LIN {X 0,Y 185.932,Z 327.325,A -85,B 0,C 180,E1 -22223.49,E2 -22223.49} C_VEL
LIN {X 0,Y 186.378,Z 327.271,A -85,B 0,C 180,E1 -22230.001,E2 -22230.001} C_VEL
LIN {X 0,Y 185.926,Z 327.327,A -85,B 0,C 180,E1 -22236.513,E2 -22236.513} C_VEL
LIN {X 0,Y 185.869,Z 327.333,A -85,B 0,C 180,E1 -22239.922,E2 -22239.922} C_VEL
LIN {X 0,Y 186.977,Z 330.337,A -85,B 0,C 180,E1 -22240.252,E2 -22240.252} C_VEL
LIN {X 0,Y 196.762,Z 352.168,A -85,B 0,C 180,E1 -22242.755,E2 -22242.755} C_VEL
LIN {X 0,Y 202.27,Z 367.616,A -85,B 0,C 180,E1 -22244.204,E2 -22244.204} C_VEL
LIN {X 0,Y 202.12,Z 374.541,A -85,B 0,C 180,E1 -22244.511,E2 -22244.511} C_VEL
LIN {X 0,Y 199.034,Z 429.376,A -85,B 0,C 180,E1 -22246.777,E2 -22246.777} C_VEL
LIN {X 0,Y 197.747,Z 443.213,A -85,B 0,C 180,E1 -22247.759,E2 -22247.759} C_VEL
LIN {X 0,Y 196.286,Z 455.635,A -85,B 0,C 180,E1 -22249.053,E2 -22249.053} C_VEL
LIN {X 0,Y 194.468,Z 467.347,A -85,B 0,C 180,E1 -22250.675,E2 -22250.675} C_VEL
LIN {X 0,Y 192.408,Z 479.143,A -85,B 0,C 180,E1 -22252.786,E2 -22252.786} C_VEL
LIN {X 0,Y 190.451,Z 489.318,A -85,B 0,C 180,E1 -22255.112,E2 -22255.112} C_VEL
LIN {X 0,Y 188.356,Z 499.162,A -85,B 0,C 180,E1 -22257.925,E2 -22257.925} C_VEL
LIN {X 0,Y 186.543,Z 507.642,A -85,B 0,C 180,E1 -22260.964,E2 -22260.964} C_VEL
LIN {X 0,Y 185.14,Z 514.465,A -85,B 0,C 180,E1 -22264.04,E2 -22264.04} C_VEL
LIN {X 0,Y 184.09,Z 520.754,A -85,B 0,C 180,E1 -22267.651,E2 -22267.651} C_VEL
LIN {X 0,Y 183.278,Z 524.854,A -85,B 0,C 180,E1 -22270.685,E2 -22270.685} C_VEL
LIN {X 0,Y 182.827,Z 528.069,A -85,B 0,C 180,E1 -22273.785,E2 -22273.785} C_VEL
LIN {X 0,Y 182.741,Z 530.438,A -85,B 0,C 180,E1 -22276.948,E2 -22276.948} C_VEL
LIN {X 0,Y 182.953,Z 531.969,A -85,B 0,C 180,E1 -22280.202,E2 -22280.202} C_VEL
LIN {X 0,Y 183.589,Z 532.61,A -85,B 0,C 180,E1 -22283.506,E2 -22283.506} C_VEL
LIN {X 0,Y 185.064,Z 532.068,A -85,B 0,C 180,E1 -22287.881,E2 -22287.881} C_VEL
LIN {X 0,Y 186.497,Z 530.891,A -85,B 0,C 180,E1 -22290.665,E2 -22290.665} C_VEL
LIN {X 0,Y 189.251,Z 527.772,A -85,B 0,C 180,E1 -22294.811,E2 -22294.811} C_VEL
LIN {X 0,Y 192.716,Z 523.296,A -85,B 0,C 180,E1 -22298.611,E2 -22298.611} C_VEL
LIN {X 0,Y 196.243,Z 518.203,A -85,B 0,C 180,E1 -22301.709,E2 -22301.709} C_VEL
LIN {X 0,Y 200.327,Z 511.596,A -85,B 0,C 180,E1 -22304.744,E2 -22304.744} C_VEL
LIN {X 0,Y 205.082,Z 503.165,A -85,B 0,C 180,E1 -22307.699,E2 -22307.699} C_VEL
LIN {X 0,Y 209.405,Z 494.509,A -85,B 0,C 180,E1 -22310.053,E2 -22310.053} C_VEL
LIN {X 0,Y 213.974,Z 483.997,A -85,B 0,C 180,E1 -22312.253,E2 -22312.253} C_VEL
LIN {X 0,Y 217.979,Z 473.293,A -85,B 0,C 180,E1 -22313.986,E2 -22313.986} C_VEL
LIN {X 0,Y 221.603,Z 461.549,A -85,B 0,C 180,E1 -22315.452,E2 -22315.452} C_VEL
LIN {X 0,Y 224.7,Z 448.564,A -85,B 0,C 180,E1 -22316.683,E2 -22316.683} C_VEL
LIN {X 0,Y 226.822,Z 436.927,A -85,B 0,C 180,E1 -22317.465,E2 -22317.465} C_VEL
LIN {X 0,Y 228.488,Z 423.317,A -85,B 0,C 180,E1 -22318.057,E2 -22318.057} C_VEL
LIN {X 0,Y 231.675,Z 389.447,A -85,B 0,C 180,E1 -22319.266,E2 -22319.266} C_VEL
LIN {X 0,Y 228.046,Z 381.272,A -85,B 0,C 180,E1 -22321.321,E2 -22321.321} C_VEL
LIN {X 0,Y 223.31,Z 372.435,A -85,B 0,C 180,E1 -22324.297,E2 -22324.297} C_VEL
LIN {X 0,Y 221.558,Z 369.535,A -85,B 0,C 180,E1 -22325.549,E2 -22325.549} C_VEL
LIN {X 0,Y 219.232,Z 366.365,A -85,B 0,C 180,E1 -22327.272,E2 -22327.272} C_VEL
LIN {X 0,Y 216.775,Z 362.911,A -85,B 0,C 180,E1 -22329.412,E2 -22329.412} C_VEL
LIN {X 0,Y 215.973,Z 361.635,A -85,B 0,C 180,E1 -22330.212,E2 -22330.212} C_VEL
LIN {X 0,Y 213.658,Z 358.637,A -85,B 0,C 180,E1 -22332.793,E2 -22332.793} C_VEL
LIN {X 0,Y 212.698,Z 357.131,A -85,B 0,C 180,E1 -22334.145,E2 -22334.145} C_VEL
LIN {X 0,Y 209.868,Z 354.113,A -85,B 0,C 180,E1 -22340.336,E2 -22340.336} C_VEL
LIN {X 0,Y 209.512,Z 354.074,A -85,B 0,C 180,E1 -22343.736,E2 -22343.736} C_VEL
LIN {X 0,Y 210.326,Z 355.309,A -85,B 0,C 180,E1 -22348.017,E2 -22348.017} C_VEL
LIN {X 0,Y 213.689,Z 361.325,A -85,B 0,C 180,E1 -22354.13,E2 -22354.13} C_VEL
LIN {X 0,Y 214.623,Z 362.828,A -85,B 0,C 180,E1 -22355.247,E2 -22355.247} C_VEL
LIN {X 0,Y 218.016,Z 368.735,A -85,B 0,C 180,E1 -22358.63,E2 -22358.63} C_VEL
LIN {X 0,Y 221.061,Z 374.393,A -85,B 0,C 180,E1 -22361.077,E2 -22361.077} C_VEL
LIN {X 0,Y 224.31,Z 380.915,A -85,B 0,C 180,E1 -22363.359,E2 -22363.359} C_VEL
LIN {X 0,Y 227.742,Z 388.861,A -85,B 0,C 180,E1 -22365.565,E2 -22365.565} C_VEL
LIN {X 0,Y 230.944,Z 397.58,A -85,B 0,C 180,E1 -22367.451,E2 -22367.451} C_VEL
LIN {X 0,Y 230.913,Z 400.519,A -85,B 0,C 180,E1 -22367.647,E2 -22367.647} C_VEL
LIN {X 0,Y 229.169,Z 419.232,A -85,B 0,C 180,E1 -22368.32,E2 -22368.32} C_VEL
LIN {X 0,Y 228.187,Z 425.066,A -85,B 0,C 180,E1 -22368.359,E2 -22368.359} C_VEL
LIN {X 0,Y 222.704,Z 444.072,A -85,B 0,C 180,E1 -22367.877,E2 -22367.877} C_VEL
LIN {X 0,Y 221.385,Z 449.752,A -85,B 0,C 180,E1 -22368.055,E2 -22368.055} C_VEL
LIN {X 0,Y 218.319,Z 463.228,A -85,B 0,C 180,E1 -22369.011,E2 -22369.011} C_VEL
LIN {X 0,Y 214.436,Z 476.108,A -85,B 0,C 180,E1 -22370.274,E2 -22370.274} C_VEL
LIN {X 0,Y 210.252,Z 487.489,A -85,B 0,C 180,E1 -22371.8,E2 -22371.8} C_VEL
LIN {X 0,Y 205.221,Z 498.939,A -85,B 0,C 180,E1 -22373.789,E2 -22373.789} C_VEL
LIN {X 0,Y 200.711,Z 508.249,A -85,B 0,C 180,E1 -22375.926,E2 -22375.926} C_VEL
LIN {X 0,Y 195.659,Z 517.339,A -85,B 0,C 180,E1 -22378.611,E2 -22378.611} C_VEL
LIN {X 0,Y 191.14,Z 524.734,A -85,B 0,C 180,E1 -22381.444,E2 -22381.444} C_VEL
LIN {X 0,Y 186.745,Z 531.404,A -85,B 0,C 180,E1 -22384.788,E2 -22384.788} C_VEL
LIN {X 0,Y 182.953,Z 536.942,A -85,B 0,C 180,E1 -22388.595,E2 -22388.595} C_VEL
LIN {X 0,Y 180.238,Z 540.388,A -85,B 0,C 180,E1 -22391.822,E2 -22391.822} C_VEL
LIN {X 0,Y 178.806,Z 542.134,A -85,B 0,C 180,E1 -22394.029,E2 -22394.029} C_VEL
LIN {X 0,Y 177.03,Z 544.467,A -85,B 0,C 180,E1 -22398.55,E2 -22398.55} C_VEL
LIN {X 0,Y 176.466,Z 545.033,A -85,B 0,C 180,E1 -22400.832,E2 -22400.832} C_VEL
LIN {X 0,Y 176.026,Z 544.984,A -85,B 0,C 180,E1 -22405.419,E2 -22405.419} C_VEL
LIN {X 0,Y 176.14,Z 544.385,A -85,B 0,C 180,E1 -22407.712,E2 -22407.712} C_VEL
LIN {X 0,Y 176.36,Z 543.376,A -85,B 0,C 180,E1 -22409.999,E2 -22409.999} C_VEL
LIN {X 0,Y 176.211,Z 541.866,A -85,B 0,C 180,E1 -22412.284,E2 -22412.284} C_VEL
LIN {X 0,Y 176.247,Z 538.77,A -85,B 0,C 180,E1 -22415.72,E2 -22415.72} C_VEL
LIN {X 0,Y 176.544,Z 534.538,A -85,B 0,C 180,E1 -22419.161,E2 -22419.161} C_VEL
LIN {X 0,Y 177.418,Z 528.024,A -85,B 0,C 180,E1 -22423.165,E2 -22423.165} C_VEL
LIN {X 0,Y 178.809,Z 520.861,A -85,B 0,C 180,E1 -22426.555,E2 -22426.555} C_VEL
LIN {X 0,Y 180.712,Z 511.856,A -85,B 0,C 180,E1 -22429.893,E2 -22429.893} C_VEL
LIN {X 0,Y 182.69,Z 502.602,A -85,B 0,C 180,E1 -22432.623,E2 -22432.623} C_VEL
LIN {X 0,Y 184.788,Z 492.337,A -85,B 0,C 180,E1 -22435.03,E2 -22435.03} C_VEL
LIN {X 0,Y 186.95,Z 481.014,A -85,B 0,C 180,E1 -22437.116,E2 -22437.116} C_VEL
LIN {X 0,Y 188.885,Z 470.453,A -85,B 0,C 180,E1 -22438.622,E2 -22438.622} C_VEL
LIN {X 0,Y 190.679,Z 457.862,A -85,B 0,C 180,E1 -22439.991,E2 -22439.991} C_VEL
LIN {X 0,Y 192.129,Z 443.75,A -85,B 0,C 180,E1 -22441.032,E2 -22441.032} C_VEL
LIN {X 0,Y 194.899,Z 391.791,A -85,B 0,C 180,E1 -22443.296,E2 -22443.296} C_VEL
LIN {X 0,Y 192.181,Z 367.369,A -85,B 0,C 180,E1 -22444.862,E2 -22444.862} C_VEL
LIN {X 0,Y 183.309,Z 342.833,A -85,B 0,C 180,E1 -22447.406,E2 -22447.406} C_VEL
LIN {X 0,Y 179.794,Z 333.815,A -85,B 0,C 180,E1 -22448.464,E2 -22448.464} C_VEL
LIN {X 0,Y 178.436,Z 328.259,A -85,B 0,C 180,E1 -22451.615,E2 -22451.615} C_VEL
LIN {X 0,Y 178.389,Z 328.264,A -85,B 0,C 180,E1 -22455.163,E2 -22455.163} C_VEL
LIN {X 0,Y 178.406,Z 328.265,A -85,B 0,C 180,E1 -22458.456,E2 -22458.456} C_VEL
LIN {X 0,Y 178.46,Z 328.256,A -85,B 0,C 180,E1 -22461.962,E2 -22461.962} C_VEL
LIN {X 0,Y 178.486,Z 328.246,A -85,B 0,C 180,E1 -22466.547,E2 -22466.547} C_VEL
LIN {X 0,Y 178.519,Z 328.222,A -85,B 0,C 180,E1 -22470.006,E2 -22470.006} C_VEL
LIN {X 0,Y 178.53,Z 328.248,A -85,B 0,C 180,E1 -22474.875,E2 -22474.875} C_VEL
LIN {X 0,Y 178.619,Z 328.23,A -85,B 0,C 180,E1 -22480.784,E2 -22480.784} C_VEL
LIN {X 0,Y 178.661,Z 328.229,A -85,B 0,C 180,E1 -22484.017,E2 -22484.017} C_VEL
LIN {X 0,Y 178.857,Z 328.195,A -85,B 0,C 180,E1 -22489.21,E2 -22489.21} C_VEL
LIN {X 0,Y 178.92,Z 328.198,A -85,B 0,C 180,E1 -22493.233,E2 -22493.233} C_VEL
LIN {X 0,Y 179.149,Z 328.155,A -85,B 0,C 180,E1 -22497.752,E2 -22497.752} C_VEL
LIN {X 0,Y 179.365,Z 328.128,A -85,B 0,C 180,E1 -22500.001,E2 -22500.001} C_VEL
LIN {X 0,Y 178.857,Z 328.202,A -85,B 0,C 180,E1 -22504.508,E2 -22504.508} C_VEL
LIN {X 0,Y 178.903,Z 328.188,A -85,B 0,C 180,E1 -22509.041,E2 -22509.041} C_VEL
LIN {X 0,Y 178.654,Z 328.215,A -85,B 0,C 180,E1 -22513.653,E2 -22513.653} C_VEL
LIN {X 0,Y 178.619,Z 328.231,A -85,B 0,C 180,E1 -22519.216,E2 -22519.216} C_VEL
LIN {X 0,Y 178.512,Z 328.224,A -85,B 0,C 180,E1 -22525.112,E2 -22525.112} C_VEL
LIN {X 0,Y 178.457,Z 328.254,A -85,B 0,C 180,E1 -22530.796,E2 -22530.796} C_VEL
LIN {X 0,Y 178.48,Z 328.252,A -85,B 0,C 180,E1 -22534.22,E2 -22534.22} C_VEL
LIN {X 0,Y 178.392,Z 328.244,A -85,B 0,C 180,E1 -22539.076,E2 -22539.076} C_VEL
LIN {X 0,Y 178.396,Z 328.251,A -85,B 0,C 180,E1 -22542.047,E2 -22542.047} C_VEL
LIN {X 0,Y 178.391,Z 328.264,A -85,B 0,C 180,E1 -22545.166,E2 -22545.166} C_VEL
LIN {X 0,Y 178.398,Z 328.261,A -85,B 0,C 180,E1 -22548.462,E2 -22548.462} C_VEL
LIN {X 0,Y 178.419,Z 328.249,A -85,B 0,C 180,E1 -22553.784,E2 -22553.784} C_VEL
LIN {X 0,Y 178.484,Z 328.249,A -85,B 0,C 180,E1 -22556.548,E2 -22556.548} C_VEL
LIN {X 0,Y 178.444,Z 328.257,A -85,B 0,C 180,E1 -22561.797,E2 -22561.797} C_VEL
LIN {X 0,Y 178.516,Z 328.246,A -85,B 0,C 180,E1 -22564.891,E2 -22564.891} C_VEL
LIN {X 0,Y 178.592,Z 328.236,A -85,B 0,C 180,E1 -22570.816,E2 -22570.816} C_VEL
LIN {X 0,Y 178.649,Z 328.23,A -85,B 0,C 180,E1 -22576.349,E2 -22576.349} C_VEL
LIN {X 0,Y 178.909,Z 328.196,A -85,B 0,C 180,E1 -22580.961,E2 -22580.961} C_VEL
LIN {X 0,Y 178.823,Z 328.211,A -85,B 0,C 180,E1 -22585.493,E2 -22585.493} C_VEL
LIN {X 0,Y 179.343,Z 328.147,A -85,B 0,C 180,E1 -22590.001,E2 -22590.001} C_VEL
LIN {X 0,Y 178.891,Z 328.204,A -85,B 0,C 180,E1 -22596.77,E2 -22596.77} C_VEL
LIN {X 0,Y 178.9,Z 328.202,A -85,B 0,C 180,E1 -22598.828,E2 -22598.828} C_VEL
LIN {X 0,Y 180.038,Z 331.288,A -85,B 0,C 180,E1 -22599.202,E2 -22599.202} C_VEL
LIN {X 0,Y 190.433,Z 354.403,A -85,B 0,C 180,E1 -22601.998,E2 -22601.998} C_VEL
LIN {X 0,Y 195.809,Z 369.321,A -85,B 0,C 180,E1 -22603.465,E2 -22603.465} C_VEL
LIN {X 0,Y 192.405,Z 429.574,A -85,B 0,C 180,E1 -22606.037,E2 -22606.037} C_VEL
LIN {X 0,Y 191.108,Z 443.163,A -85,B 0,C 180,E1 -22607.027,E2 -22607.027} C_VEL
LIN {X 0,Y 189.571,Z 455.754,A -85,B 0,C 180,E1 -22608.369,E2 -22608.369} C_VEL
LIN {X 0,Y 187.535,Z 468.499,A -85,B 0,C 180,E1 -22610.211,E2 -22610.211} C_VEL
LIN {X 0,Y 185.541,Z 479.448,A -85,B 0,C 180,E1 -22612.26,E2 -22612.26} C_VEL
LIN {X 0,Y 183.567,Z 489.367,A -85,B 0,C 180,E1 -22614.604,E2 -22614.604} C_VEL
LIN {X 0,Y 181.237,Z 499.888,A -85,B 0,C 180,E1 -22617.733,E2 -22617.733} C_VEL
LIN {X 0,Y 179.555,Z 507.536,A -85,B 0,C 180,E1 -22620.588,E2 -22620.588} C_VEL
LIN {X 0,Y 178.014,Z 514.825,A -85,B 0,C 180,E1 -22623.994,E2 -22623.994} C_VEL
LIN {X 0,Y 177.021,Z 520.623,A -85,B 0,C 180,E1 -22627.435,E2 -22627.435} C_VEL
LIN {X 0,Y 176.009,Z 526.046,A -85,B 0,C 180,E1 -22631.672,E2 -22631.672} C_VEL
LIN {X 0,Y 175.708,Z 528.231,A -85,B 0,C 180,E1 -22633.947,E2 -22633.947} C_VEL
LIN {X 0,Y 175.64,Z 530.583,A -85,B 0,C 180,E1 -22637.137,E2 -22637.137} C_VEL
LIN {X 0,Y 175.864,Z 532.059,A -85,B 0,C 180,E1 -22640.252,E2 -22640.252} C_VEL
LIN {X 0,Y 176.433,Z 532.801,A -85,B 0,C 180,E1 -22643.308,E2 -22643.308} C_VEL
LIN {X 0,Y 177.347,Z 532.862,A -85,B 0,C 180,E1 -22646.327,E2 -22646.327} C_VEL
LIN {X 0,Y 178.845,Z 532.021,A -85,B 0,C 180,E1 -22649.83,E2 -22649.83} C_VEL
LIN {X 0,Y 180.926,Z 530.19,A -85,B 0,C 180,E1 -22653.309,E2 -22653.309} C_VEL
LIN {X 0,Y 184.378,Z 526.376,A -85,B 0,C 180,E1 -22657.593,E2 -22657.593} C_VEL
LIN {X 0,Y 188.575,Z 521.072,A -85,B 0,C 180,E1 -22661.531,E2 -22661.531} C_VEL
LIN {X 0,Y 192.796,Z 515.008,A -85,B 0,C 180,E1 -22664.778,E2 -22664.778} C_VEL
LIN {X 0,Y 197.313,Z 507.876,A -85,B 0,C 180,E1 -22667.66,E2 -22667.66} C_VEL
LIN {X 0,Y 201.369,Z 500.691,A -85,B 0,C 180,E1 -22669.95,E2 -22669.95} C_VEL
LIN {X 0,Y 206.231,Z 491.061,A -85,B 0,C 180,E1 -22672.353,E2 -22672.353} C_VEL
LIN {X 0,Y 210.917,Z 480.235,A -85,B 0,C 180,E1 -22674.438,E2 -22674.438} C_VEL
LIN {X 0,Y 214.966,Z 469.363,A -85,B 0,C 180,E1 -22676.031,E2 -22676.031} C_VEL
LIN {X 0,Y 218.614,Z 457.119,A -85,B 0,C 180,E1 -22677.428,E2 -22677.428} C_VEL
LIN {X 0,Y 221.428,Z 444.49,A -85,B 0,C 180,E1 -22678.499,E2 -22678.499} C_VEL
LIN {X 0,Y 223.678,Z 430.863,A -85,B 0,C 180,E1 -22679.264,E2 -22679.264} C_VEL
LIN {X 0,Y 227.534,Z 392.525,A -85,B 0,C 180,E1 -22680.653,E2 -22680.653} C_VEL
LIN {X 0,Y 224.843,Z 386.263,A -85,B 0,C 180,E1 -22682.345,E2 -22682.345} C_VEL
LIN {X 0,Y 220.675,Z 378.083,A -85,B 0,C 180,E1 -22685.189,E2 -22685.189} C_VEL
LIN {X 0,Y 218.785,Z 375.043,A -85,B 0,C 180,E1 -22686.615,E2 -22686.615} C_VEL
LIN {X 0,Y 216.996,Z 372.54,A -85,B 0,C 180,E1 -22688.042,E2 -22688.042} C_VEL
LIN {X 0,Y 214.581,Z 368.698,A -85,B 0,C 180,E1 -22690.381,E2 -22690.381} C_VEL
LIN {X 0,Y 212.013,Z 365.144,A -85,B 0,C 180,E1 -22693.417,E2 -22693.417} C_VEL
LIN {X 0,Y 211.324,Z 364.026,A -85,B 0,C 180,E1 -22694.437,E2 -22694.437} C_VEL
LIN {X 0,Y 208.679,Z 361.081,A -85,B 0,C 180,E1 -22700.638,E2 -22700.638} C_VEL
LIN {X 0,Y 208.431,Z 361.217,A -85,B 0,C 180,E1 -22704.437,E2 -22704.437} C_VEL
LIN {X 0,Y 209.088,Z 362.272,A -85,B 0,C 180,E1 -22707.757,E2 -22707.757} C_VEL
LIN {X 0,Y 212.476,Z 368.477,A -85,B 0,C 180,E1 -22714.099,E2 -22714.099} C_VEL
LIN {X 0,Y 215.891,Z 374.87,A -85,B 0,C 180,E1 -22717.868,E2 -22717.868} C_VEL
LIN {X 0,Y 218.569,Z 380.161,A -85,B 0,C 180,E1 -22720.209,E2 -22720.209} C_VEL
LIN {X 0,Y 221.832,Z 387.124,A -85,B 0,C 180,E1 -22722.696,E2 -22722.696} C_VEL
LIN {X 0,Y 224.798,Z 394.55,A -85,B 0,C 180,E1 -22724.738,E2 -22724.738} C_VEL
LIN {X 0,Y 226.974,Z 400.826,A -85,B 0,C 180,E1 -22726.157,E2 -22726.157} C_VEL
LIN {X 0,Y 222.767,Z 441.68,A -85,B 0,C 180,E1 -22727.656,E2 -22727.656} C_VEL
LIN {X 0,Y 221.385,Z 449.752,A -85,B 0,C 180,E1 -22728.055,E2 -22728.055} C_VEL
LIN {X 0,Y 219.871,Z 455.421,A -85,B 0,C 180,E1 -22728.258,E2 -22728.258} C_VEL
LIN {X 0,Y 215.922,Z 464.53,A -85,B 0,C 180,E1 -22728.339,E2 -22728.339} C_VEL
LIN {X 0,Y 211.504,Z 473.339,A -85,B 0,C 180,E1 -22728.57,E2 -22728.57} C_VEL
LIN {X 0,Y 209.263,Z 478.531,A -85,B 0,C 180,E1 -22729.019,E2 -22729.019} C_VEL
LIN {X 0,Y 204.813,Z 489.681,A -85,B 0,C 180,E1 -22730.593,E2 -22730.593} C_VEL
LIN {X 0,Y 199.645,Z 500.607,A -85,B 0,C 180,E1 -22732.608,E2 -22732.608} C_VEL
LIN {X 0,Y 194.03,Z 511.085,A -85,B 0,C 180,E1 -22735.215,E2 -22735.215} C_VEL
LIN {X 0,Y 189.699,Z 518.281,A -85,B 0,C 180,E1 -22737.506,E2 -22737.506} C_VEL
LIN {X 0,Y 184.989,Z 525.47,A -85,B 0,C 180,E1 -22740.402,E2 -22740.402} C_VEL
LIN {X 0,Y 180.201,Z 532.11,A -85,B 0,C 180,E1 -22743.975,E2 -22743.975} C_VEL
LIN {X 0,Y 176.367,Z 537.202,A -85,B 0,C 180,E1 -22747.754,E2 -22747.754} C_VEL
LIN {X 0,Y 173.491,Z 540.49,A -85,B 0,C 180,E1 -22751.089,E2 -22751.089} C_VEL
LIN {X 0,Y 171.966,Z 542.167,A -85,B 0,C 180,E1 -22753.375,E2 -22753.375} C_VEL
LIN {X 0,Y 170.863,Z 543.452,A -85,B 0,C 180,E1 -22755.711,E2 -22755.711} C_VEL
LIN {X 0,Y 169.449,Z 544.793,A -85,B 0,C 180,E1 -22760.449,E2 -22760.449} C_VEL
LIN {X 0,Y 168.939,Z 544.618,A -85,B 0,C 180,E1 -22765.226,E2 -22765.226} C_VEL
LIN {X 0,Y 169.054,Z 543.945,A -85,B 0,C 180,E1 -22767.616,E2 -22767.616} C_VEL
LIN {X 0,Y 169.297,Z 542.827,A -85,B 0,C 180,E1 -22769.999,E2 -22769.999} C_VEL
LIN {X 0,Y 169.15,Z 539.642,A -85,B 0,C 180,E1 -22774.31,E2 -22774.31} C_VEL
LIN {X 0,Y 169.362,Z 535.249,A -85,B 0,C 180,E1 -22778.35,E2 -22778.35} C_VEL
LIN {X 0,Y 170.148,Z 529.021,A -85,B 0,C 180,E1 -22782.523,E2 -22782.523} C_VEL
LIN {X 0,Y 171.405,Z 522.168,A -85,B 0,C 180,E1 -22786.066,E2 -22786.066} C_VEL
LIN {X 0,Y 173.245,Z 513.616,A -85,B 0,C 180,E1 -22789.551,E2 -22789.551} C_VEL
LIN {X 0,Y 175.336,Z 504.105,A -85,B 0,C 180,E1 -22792.59,E2 -22792.59} C_VEL
LIN {X 0,Y 177.528,Z 493.903,A -85,B 0,C 180,E1 -22795.185,E2 -22795.185} C_VEL
LIN {X 0,Y 179.721,Z 483.092,A -85,B 0,C 180,E1 -22797.352,E2 -22797.352} C_VEL
LIN {X 0,Y 181.998,Z 471.178,A -85,B 0,C 180,E1 -22799.176,E2 -22799.176} C_VEL
LIN {X 0,Y 183.803,Z 458.939,A -85,B 0,C 180,E1 -22800.597,E2 -22800.597} C_VEL
LIN {X 0,Y 185.356,Z 445.7,A -85,B 0,C 180,E1 -22801.66,E2 -22801.66} C_VEL
LIN {X 0,Y 186.511,Z 425.843,A -85,B 0,C 180,E1 -22802.649,E2 -22802.649} C_VEL
LIN {X 0,Y 188.343,Z 392.052,A -85,B 0,C 180,E1 -22804.131,E2 -22804.131} C_VEL
LIN {X 0,Y 185.794,Z 369.391,A -85,B 0,C 180,E1 -22805.633,E2 -22805.633} C_VEL
LIN {X 0,Y 177.448,Z 346.002,A -85,B 0,C 180,E1 -22808.165,E2 -22808.165} C_VEL
LIN {X 0,Y 172.399,Z 333.413,A -85,B 0,C 180,E1 -22809.804,E2 -22809.804} C_VEL
LIN {X 0,Y 171.345,Z 329.142,A -85,B 0,C 180,E1 -22812.414,E2 -22812.414} C_VEL
LIN {X 0,Y 171.335,Z 329.144,A -85,B 0,C 180,E1 -22817.588,E2 -22817.588} C_VEL
LIN {X 0,Y 171.409,Z 329.134,A -85,B 0,C 180,E1 -22822.047,E2 -22822.047} C_VEL
LIN {X 0,Y 171.403,Z 329.133,A -85,B 0,C 180,E1 -22825.087,E2 -22825.087} C_VEL
LIN {X 0,Y 171.445,Z 329.105,A -85,B 0,C 180,E1 -22830.534,E2 -22830.534} C_VEL
LIN {X 0,Y 171.454,Z 329.13,A -85,B 0,C 180,E1 -22835.801,E2 -22835.801} C_VEL
LIN {X 0,Y 171.575,Z 329.107,A -85,B 0,C 180,E1 -22840.872,E2 -22840.872} C_VEL
LIN {X 0,Y 171.605,Z 329.105,A -85,B 0,C 180,E1 -22845.776,E2 -22845.776} C_VEL
LIN {X 0,Y 171.884,Z 329.069,A -85,B 0,C 180,E1 -22850.587,E2 -22850.587} C_VEL
LIN {X 0,Y 171.817,Z 329.08,A -85,B 0,C 180,E1 -22855.308,E2 -22855.308} C_VEL
LIN {X 0,Y 172.328,Z 329.004,A -85,B 0,C 180,E1 -22860.001,E2 -22860.001} C_VEL
LIN {X 0,Y 171.805,Z 329.08,A -85,B 0,C 180,E1 -22864.693,E2 -22864.693} C_VEL
LIN {X 0,Y 171.84,Z 329.066,A -85,B 0,C 180,E1 -22869.416,E2 -22869.416} C_VEL
LIN {X 0,Y 171.572,Z 329.1,A -85,B 0,C 180,E1 -22874.228,E2 -22874.228} C_VEL
LIN {X 0,Y 171.538,Z 329.113,A -85,B 0,C 180,E1 -22879.56,E2 -22879.56} C_VEL
LIN {X 0,Y 171.44,Z 329.103,A -85,B 0,C 180,E1 -22885.6,E2 -22885.6} C_VEL
LIN {X 0,Y 171.414,Z 329.13,A -85,B 0,C 180,E1 -22890.574,E2 -22890.574} C_VEL
LIN {X 0,Y 171.39,Z 329.132,A -85,B 0,C 180,E1 -22895.036,E2 -22895.036} C_VEL
LIN {X 0,Y 171.355,Z 329.121,A -85,B 0,C 180,E1 -22898.809,E2 -22898.809} C_VEL
LIN {X 0,Y 171.318,Z 329.14,A -85,B 0,C 180,E1 -22904.219,E2 -22904.219} C_VEL
LIN {X 0,Y 171.33,Z 329.14,A -85,B 0,C 180,E1 -22908.982,E2 -22908.982} C_VEL
LIN {X 0,Y 171.36,Z 329.124,A -85,B 0,C 180,E1 -22912.036,E2 -22912.036} C_VEL
LIN {X 0,Y 171.397,Z 329.128,A -85,B 0,C 180,E1 -22915.095,E2 -22915.095} C_VEL
LIN {X 0,Y 171.409,Z 329.13,A -85,B 0,C 180,E1 -22920.529,E2 -22920.529} C_VEL
LIN {X 0,Y 171.442,Z 329.128,A -85,B 0,C 180,E1 -22925.801,E2 -22925.801} C_VEL
LIN {X 0,Y 171.548,Z 329.114,A -85,B 0,C 180,E1 -22930.87,E2 -22930.87} C_VEL
LIN {X 0,Y 171.564,Z 329.115,A -85,B 0,C 180,E1 -22935.773,E2 -22935.773} C_VEL
LIN {X 0,Y 171.847,Z 329.076,A -85,B 0,C 180,E1 -22940.586,E2 -22940.586} C_VEL
LIN {X 0,Y 171.774,Z 329.089,A -85,B 0,C 180,E1 -22945.308,E2 -22945.308} C_VEL
LIN {X 0,Y 172.308,Z 329.023,A -85,B 0,C 180,E1 -22950.001,E2 -22950.001} C_VEL
LIN {X 0,Y 171.862,Z 329.079,A -85,B 0,C 180,E1 -22957.048,E2 -22957.048} C_VEL
LIN {X 0,Y 171.865,Z 329.078,A -85,B 0,C 180,E1 -22957.639,E2 -22957.639} C_VEL
LIN {X 0,Y 172.906,Z 331.993,A -85,B 0,C 180,E1 -22958.033,E2 -22958.033} C_VEL
LIN {X 0,Y 183.085,Z 354.229,A -85,B 0,C 180,E1 -22960.927,E2 -22960.927} C_VEL
LIN {X 0,Y 187.981,Z 366.948,A -85,B 0,C 180,E1 -22962.296,E2 -22962.296} C_VEL
LIN {X 0,Y 189.272,Z 370.814,A -85,B 0,C 180,E1 -22962.669,E2 -22962.669} C_VEL
LIN {X 0,Y 185.823,Z 429.182,A -85,B 0,C 180,E1 -22965.238,E2 -22965.238} C_VEL
LIN {X 0,Y 184.501,Z 442.645,A -85,B 0,C 180,E1 -22966.233,E2 -22966.233} C_VEL
LIN {X 0,Y 182.876,Z 455.757,A -85,B 0,C 180,E1 -22967.659,E2 -22967.659} C_VEL
LIN {X 0,Y 180.746,Z 468.739,A -85,B 0,C 180,E1 -22969.596,E2 -22969.596} C_VEL
LIN {X 0,Y 178.749,Z 479.295,A -85,B 0,C 180,E1 -22971.631,E2 -22971.631} C_VEL
LIN {X 0,Y 176.436,Z 490.374,A -85,B 0,C 180,E1 -22974.354,E2 -22974.354} C_VEL
LIN {X 0,Y 174.191,Z 500.238,A -85,B 0,C 180,E1 -22977.422,E2 -22977.422} C_VEL
LIN {X 0,Y 172.407,Z 508.197,A -85,B 0,C 180,E1 -22980.53,E2 -22980.53} C_VEL
LIN {X 0,Y 170.892,Z 515.223,A -85,B 0,C 180,E1 -22983.976,E2 -22983.976} C_VEL
LIN {X 0,Y 169.912,Z 520.763,A -85,B 0,C 180,E1 -22987.392,E2 -22987.392} C_VEL
LIN {X 0,Y 168.881,Z 526.157,A -85,B 0,C 180,E1 -22991.748,E2 -22991.748} C_VEL
LIN {X 0,Y 168.545,Z 529.198,A -85,B 0,C 180,E1 -22995.144,E2 -22995.144} C_VEL
LIN {X 0,Y 168.59,Z 531.387,A -85,B 0,C 180,E1 -22998.624,E2 -22998.624} C_VEL
LIN {X 0,Y 169.055,Z 532.733,A -85,B 0,C 180,E1 -23002.175,E2 -23002.175} C_VEL
LIN {X 0,Y 170.006,Z 533.205,A -85,B 0,C 180,E1 -23005.773,E2 -23005.773} C_VEL
LIN {X 0,Y 171.471,Z 532.756,A -85,B 0,C 180,E1 -23009.399,E2 -23009.399} C_VEL
LIN {X 0,Y 173.909,Z 530.981,A -85,B 0,C 180,E1 -23013.606,E2 -23013.606} C_VEL
LIN {X 0,Y 177.376,Z 527.65,A -85,B 0,C 180,E1 -23017.935,E2 -23017.935} C_VEL
LIN {X 0,Y 180.513,Z 524.126,A -85,B 0,C 180,E1 -23021.006,E2 -23021.006} C_VEL
LIN {X 0,Y 185.011,Z 518.538,A -85,B 0,C 180,E1 -23024.578,E2 -23024.578} C_VEL
LIN {X 0,Y 189.682,Z 511.92,A -85,B 0,C 180,E1 -23027.698,E2 -23027.698} C_VEL
LIN {X 0,Y 194.964,Z 503.534,A -85,B 0,C 180,E1 -23030.709,E2 -23030.709} C_VEL
LIN {X 0,Y 200.148,Z 494.2,A -85,B 0,C 180,E1 -23033.248,E2 -23033.248} C_VEL
LIN {X 0,Y 205.148,Z 483.747,A -85,B 0,C 180,E1 -23035.42,E2 -23035.42} C_VEL
LIN {X 0,Y 209.263,Z 473.703,A -85,B 0,C 180,E1 -23037.036,E2 -23037.036} C_VEL
LIN {X 0,Y 213.146,Z 462.261,A -85,B 0,C 180,E1 -23038.464,E2 -23038.464} C_VEL
LIN {X 0,Y 216.378,Z 449.933,A -85,B 0,C 180,E1 -23039.651,E2 -23039.651} C_VEL
LIN {X 0,Y 218.747,Z 438.372,A -85,B 0,C 180,E1 -23040.438,E2 -23040.438} C_VEL
LIN {X 0,Y 220.619,Z 424.835,A -85,B 0,C 180,E1 -23041.05,E2 -23041.05} C_VEL
LIN {X 0,Y 223.628,Z 395.667,A -85,B 0,C 180,E1 -23042.11,E2 -23042.11} C_VEL
LIN {X 0,Y 221.2,Z 390.204,A -85,B 0,C 180,E1 -23043.747,E2 -23043.747} C_VEL
LIN {X 0,Y 218.098,Z 383.718,A -85,B 0,C 180,E1 -23046.107,E2 -23046.107} C_VEL
LIN {X 0,Y 215.57,Z 379.634,A -85,B 0,C 180,E1 -23048.184,E2 -23048.184} C_VEL
LIN {X 0,Y 212.889,Z 375.499,A -85,B 0,C 180,E1 -23050.831,E2 -23050.831} C_VEL
LIN {X 0,Y 209.956,Z 370.918,A -85,B 0,C 180,E1 -23054.733,E2 -23054.733} C_VEL
LIN {X 0,Y 207.529,Z 368.077,A -85,B 0,C 180,E1 -23060.757,E2 -23060.757} C_VEL
LIN {X 0,Y 207.394,Z 368.384,A -85,B 0,C 180,E1 -23065.216,E2 -23065.216} C_VEL
LIN {X 0,Y 207.826,Z 369.16,A -85,B 0,C 180,E1 -23067.393,E2 -23067.393} C_VEL
LIN {X 0,Y 210.884,Z 375.122,A -85,B 0,C 180,E1 -23073.574,E2 -23073.574} C_VEL
LIN {X 0,Y 213.841,Z 381.07,A -85,B 0,C 180,E1 -23077.12,E2 -23077.12} C_VEL
LIN {X 0,Y 216.32,Z 386.353,A -85,B 0,C 180,E1 -23079.493,E2 -23079.493} C_VEL
LIN {X 0,Y 219.173,Z 392.923,A -85,B 0,C 180,E1 -23081.859,E2 -23081.859} C_VEL
LIN {X 0,Y 221.823,Z 399.909,A -85,B 0,C 180,E1 -23083.814,E2 -23083.814} C_VEL
LIN {X 0,Y 223.044,Z 403.645,A -85,B 0,C 180,E1 -23084.698,E2 -23084.698} C_VEL
LIN {X 0,Y 219.002,Z 440.931,A -85,B 0,C 180,E1 -23086.083,E2 -23086.083} C_VEL
LIN {X 0,Y 216.412,Z 454.442,A -85,B 0,C 180,E1 -23086.805,E2 -23086.805} C_VEL
LIN {X 0,Y 213.141,Z 466.958,A -85,B 0,C 180,E1 -23087.79,E2 -23087.79} C_VEL
LIN {X 0,Y 209.263,Z 478.531,A -85,B 0,C 180,E1 -23089.019,E2 -23089.019} C_VEL
LIN {X 0,Y 206.87,Z 483.704,A -85,B 0,C 180,E1 -23089.535,E2 -23089.535} C_VEL
LIN {X 0,Y 201.542,Z 491.876,A -85,B 0,C 180,E1 -23090.134,E2 -23090.134} C_VEL
LIN {X 0,Y 196.024,Z 499.521,A -85,B 0,C 180,E1 -23090.919,E2 -23090.919} C_VEL
LIN {X 0,Y 193.303,Z 503.849,A -85,B 0,C 180,E1 -23091.741,E2 -23091.741} C_VEL
LIN {X 0,Y 187.406,Z 513.808,A -85,B 0,C 180,E1 -23094.459,E2 -23094.459} C_VEL
LIN {X 0,Y 182.108,Z 521.731,A -85,B 0,C 180,E1 -23097.295,E2 -23097.295} C_VEL
LIN {X 0,Y 177.36,Z 528.167,A -85,B 0,C 180,E1 -23100.308,E2 -23100.308} C_VEL
LIN {X 0,Y 173.224,Z 533.391,A -85,B 0,C 180,E1 -23103.493,E2 -23103.493} C_VEL
LIN {X 0,Y 169.804,Z 537.503,A -85,B 0,C 180,E1 -23106.845,E2 -23106.845} C_VEL
LIN {X 0,Y 166.781,Z 540.621,A -85,B 0,C 180,E1 -23110.298,E2 -23110.298} C_VEL
LIN {X 0,Y 165.157,Z 542.203,A -85,B 0,C 180,E1 -23112.669,E2 -23112.669} C_VEL
LIN {X 0,Y 163.094,Z 544.145,A -85,B 0,C 180,E1 -23117.556,E2 -23117.556} C_VEL
LIN {X 0,Y 162.023,Z 544.588,A -85,B 0,C 180,E1 -23122.522,E2 -23122.522} C_VEL
LIN {X 0,Y 161.912,Z 543.749,A -85,B 0,C 180,E1 -23126.701,E2 -23126.701} C_VEL
LIN {X 0,Y 162.233,Z 542.263,A -85,B 0,C 180,E1 -23129.999,E2 -23129.999} C_VEL
LIN {X 0,Y 162.065,Z 539.266,A -85,B 0,C 180,E1 -23134.132,E2 -23134.132} C_VEL
LIN {X 0,Y 162.209,Z 535.867,A -85,B 0,C 180,E1 -23137.467,E2 -23137.467} C_VEL
LIN {X 0,Y 162.736,Z 530.919,A -85,B 0,C 180,E1 -23141.205,E2 -23141.205} C_VEL
LIN {X 0,Y 163.757,Z 524.625,A -85,B 0,C 180,E1 -23144.92,E2 -23144.92} C_VEL
LIN {X 0,Y 165.488,Z 516.747,A -85,B 0,C 180,E1 -23148.571,E2 -23148.571} C_VEL
LIN {X 0,Y 167.283,Z 508.636,A -85,B 0,C 180,E1 -23151.567,E2 -23151.567} C_VEL
LIN {X 0,Y 169.56,Z 498.76,A -85,B 0,C 180,E1 -23154.485,E2 -23154.485} C_VEL
LIN {X 0,Y 172,Z 487.8,A -85,B 0,C 180,E1 -23157.036,E2 -23157.036} C_VEL
LIN {X 0,Y 174.093,Z 477.126,A -85,B 0,C 180,E1 -23158.973,E2 -23158.973} C_VEL
LIN {X 0,Y 176.243,Z 464.503,A -85,B 0,C 180,E1 -23160.723,E2 -23160.723} C_VEL
LIN {X 0,Y 178.059,Z 451.315,A -85,B 0,C 180,E1 -23162.029,E2 -23162.029} C_VEL
LIN {X 0,Y 179.231,Z 438.42,A -85,B 0,C 180,E1 -23162.875,E2 -23162.875} C_VEL
LIN {X 0,Y 181.838,Z 393.099,A -85,B 0,C 180,E1 -23164.942,E2 -23164.942} C_VEL
LIN {X 0,Y 179.527,Z 371.664,A -85,B 0,C 180,E1 -23166.422,E2 -23166.422} C_VEL
LIN {X 0,Y 171.233,Z 348.232,A -85,B 0,C 180,E1 -23169.082,E2 -23169.082} C_VEL
LIN {X 0,Y 165.062,Z 333.165,A -85,B 0,C 180,E1 -23171.142,E2 -23171.142} C_VEL
LIN {X 0,Y 164.289,Z 330.021,A -85,B 0,C 180,E1 -23173.19,E2 -23173.19} C_VEL
LIN {X 0,Y 164.288,Z 330.018,A -85,B 0,C 180,E1 -23176.808,E2 -23176.808} C_VEL
LIN {X 0,Y 164.301,Z 330.02,A -85,B 0,C 180,E1 -23180.347,E2 -23180.347} C_VEL
LIN {X 0,Y 164.337,Z 330.014,A -85,B 0,C 180,E1 -23184.343,E2 -23184.343} C_VEL
LIN {X 0,Y 164.387,Z 329.981,A -85,B 0,C 180,E1 -23189.134,E2 -23189.134} C_VEL
LIN {X 0,Y 164.412,Z 330.006,A -85,B 0,C 180,E1 -23194.694,E2 -23194.694} C_VEL
LIN {X 0,Y 164.48,Z 329.99,A -85,B 0,C 180,E1 -23200.051,E2 -23200.051} C_VEL
LIN {X 0,Y 164.549,Z 329.987,A -85,B 0,C 180,E1 -23205.152,E2 -23205.152} C_VEL
LIN {X 0,Y 164.823,Z 329.949,A -85,B 0,C 180,E1 -23210.18,E2 -23210.18} C_VEL
LIN {X 0,Y 164.847,Z 329.949,A -85,B 0,C 180,E1 -23212.652,E2 -23212.652} C_VEL
LIN {X 0,Y 165.045,Z 329.912,A -85,B 0,C 180,E1 -23217.56,E2 -23217.56} C_VEL
LIN {X 0,Y 165.29,Z 329.879,A -85,B 0,C 180,E1 -23220.001,E2 -23220.001} C_VEL
LIN {X 0,Y 164.754,Z 329.958,A -85,B 0,C 180,E1 -23224.895,E2 -23224.895} C_VEL
LIN {X 0,Y 164.822,Z 329.948,A -85,B 0,C 180,E1 -23227.35,E2 -23227.35} C_VEL
LIN {X 0,Y 164.698,Z 329.946,A -85,B 0,C 180,E1 -23231.061,E2 -23231.061} C_VEL
LIN {X 0,Y 164.48,Z 329.991,A -85,B 0,C 180,E1 -23237.404,E2 -23237.404} C_VEL
LIN {X 0,Y 164.469,Z 329.995,A -85,B 0,C 180,E1 -23239.99,E2 -23239.99} C_VEL
LIN {X 0,Y 164.367,Z 329.985,A -85,B 0,C 180,E1 -23246.118,E2 -23246.118} C_VEL
LIN {X 0,Y 164.354,Z 330.01,A -85,B 0,C 180,E1 -23251.219,E2 -23251.219} C_VEL
LIN {X 0,Y 164.292,Z 330.011,A -85,B 0,C 180,E1 -23256.791,E2 -23256.791} C_VEL
LIN {X 0,Y 164.288,Z 329.997,A -85,B 0,C 180,E1 -23259.918,E2 -23259.918} C_VEL
LIN {X 0,Y 164.278,Z 330.015,A -85,B 0,C 180,E1 -23263.344,E2 -23263.344} C_VEL
LIN {X 0,Y 164.26,Z 330.024,A -85,B 0,C 180,E1 -23266.8,E2 -23266.8} C_VEL
LIN {X 0,Y 164.289,Z 330.013,A -85,B 0,C 180,E1 -23270.356,E2 -23270.356} C_VEL
LIN {X 0,Y 164.325,Z 330.006,A -85,B 0,C 180,E1 -23274.353,E2 -23274.353} C_VEL
LIN {X 0,Y 164.371,Z 330.011,A -85,B 0,C 180,E1 -23279.132,E2 -23279.132} C_VEL
LIN {X 0,Y 164.395,Z 330.005,A -85,B 0,C 180,E1 -23284.692,E2 -23284.692} C_VEL
LIN {X 0,Y 164.441,Z 329.999,A -85,B 0,C 180,E1 -23290.096,E2 -23290.096} C_VEL
LIN {X 0,Y 164.491,Z 329.993,A -85,B 0,C 180,E1 -23295.148,E2 -23295.148} C_VEL
LIN {X 0,Y 164.768,Z 329.959,A -85,B 0,C 180,E1 -23300.178,E2 -23300.178} C_VEL
LIN {X 0,Y 164.822,Z 329.954,A -85,B 0,C 180,E1 -23302.652,E2 -23302.652} C_VEL
LIN {X 0,Y 165.272,Z 329.9,A -85,B 0,C 180,E1 -23310.001,E2 -23310.001} C_VEL
LIN {X 0,Y 164.791,Z 330.04,A -85,B 0,C 180,E1 -23316.429,E2 -23316.429} C_VEL
LIN {X 0,Y 165.858,Z 332.875,A -85,B 0,C 180,E1 -23316.808,E2 -23316.808} C_VEL
LIN {X 0,Y 172.246,Z 346.255,A -85,B 0,C 180,E1 -23318.743,E2 -23318.743} C_VEL
LIN {X 0,Y 179.77,Z 363.765,A -85,B 0,C 180,E1 -23320.934,E2 -23320.934} C_VEL
LIN {X 0,Y 182.693,Z 372.295,A -85,B 0,C 180,E1 -23321.828,E2 -23321.828} C_VEL
LIN {X 0,Y 179.137,Z 430.282,A -85,B 0,C 180,E1 -23324.485,E2 -23324.485} C_VEL
LIN {X 0,Y 177.826,Z 443.066,A -85,B 0,C 180,E1 -23325.474,E2 -23325.474} C_VEL
LIN {X 0,Y 176.173,Z 455.957,A -85,B 0,C 180,E1 -23326.925,E2 -23326.925} C_VEL
LIN {X 0,Y 174.059,Z 468.488,A -85,B 0,C 180,E1 -23328.847,E2 -23328.847} C_VEL
LIN {X 0,Y 171.958,Z 479.171,A -85,B 0,C 180,E1 -23330.958,E2 -23330.958} C_VEL
LIN {X 0,Y 169.723,Z 489.659,A -85,B 0,C 180,E1 -23333.583,E2 -23333.583} C_VEL
LIN {X 0,Y 167.312,Z 499.91,A -85,B 0,C 180,E1 -23336.845,E2 -23336.845} C_VEL
LIN {X 0,Y 165.512,Z 507.648,A -85,B 0,C 180,E1 -23339.93,E2 -23339.93} C_VEL
LIN {X 0,Y 164.004,Z 514.384,A -85,B 0,C 180,E1 -23343.252,E2 -23343.252} C_VEL
LIN {X 0,Y 162.862,Z 520.641,A -85,B 0,C 180,E1 -23347.169,E2 -23347.169} C_VEL
LIN {X 0,Y 161.966,Z 524.958,A -85,B 0,C 180,E1 -23350.609,E2 -23350.609} C_VEL
LIN {X 0,Y 161.496,Z 528.362,A -85,B 0,C 180,E1 -23354.132,E2 -23354.132} C_VEL
LIN {X 0,Y 161.548,Z 531.692,A -85,B 0,C 180,E1 -23359.264,E2 -23359.264} C_VEL
LIN {X 0,Y 162.026,Z 532.948,A -85,B 0,C 180,E1 -23362.607,E2 -23362.607} C_VEL
LIN {X 0,Y 162.931,Z 533.481,A -85,B 0,C 180,E1 -23365.891,E2 -23365.891} C_VEL
LIN {X 0,Y 164.144,Z 533.308,A -85,B 0,C 180,E1 -23369.082,E2 -23369.082} C_VEL
LIN {X 0,Y 166.091,Z 532.312,A -85,B 0,C 180,E1 -23372.699,E2 -23372.699} C_VEL
LIN {X 0,Y 168.71,Z 530.3,A -85,B 0,C 180,E1 -23376.416,E2 -23376.416} C_VEL
LIN {X 0,Y 172.008,Z 527.238,A -85,B 0,C 180,E1 -23380.012,E2 -23380.012} C_VEL
LIN {X 0,Y 176.375,Z 522.541,A -85,B 0,C 180,E1 -23383.803,E2 -23383.803} C_VEL
LIN {X 0,Y 181.356,Z 516.476,A -85,B 0,C 180,E1 -23387.355,E2 -23387.355} C_VEL
LIN {X 0,Y 186.021,Z 510.142,A -85,B 0,C 180,E1 -23390.13,E2 -23390.13} C_VEL
LIN {X 0,Y 191.236,Z 502.044,A -85,B 0,C 180,E1 -23392.873,E2 -23392.873} C_VEL
LIN {X 0,Y 196.691,Z 492.448,A -85,B 0,C 180,E1 -23395.345,E2 -23395.345} C_VEL
LIN {X 0,Y 201.378,Z 482.934,A -85,B 0,C 180,E1 -23397.249,E2 -23397.249} C_VEL
LIN {X 0,Y 206.208,Z 471.364,A -85,B 0,C 180,E1 -23399.023,E2 -23399.023} C_VEL
LIN {X 0,Y 210.396,Z 458.91,A -85,B 0,C 180,E1 -23400.478,E2 -23400.478} C_VEL
LIN {X 0,Y 213.567,Z 446.427,A -85,B 0,C 180,E1 -23401.563,E2 -23401.563} C_VEL
LIN {X 0,Y 216.107,Z 432.749,A -85,B 0,C 180,E1 -23402.357,E2 -23402.357} C_VEL
LIN {X 0,Y 219.936,Z 398.992,A -85,B 0,C 180,E1 -23403.585,E2 -23403.585} C_VEL
LIN {X 0,Y 215.896,Z 390.011,A -85,B 0,C 180,E1 -23406.774,E2 -23406.774} C_VEL
LIN {X 0,Y 213.516,Z 385.926,A -85,B 0,C 180,E1 -23408.897,E2 -23408.897} C_VEL
LIN {X 0,Y 210.623,Z 381.302,A -85,B 0,C 180,E1 -23412.017,E2 -23412.017} C_VEL
LIN {X 0,Y 208.433,Z 377.67,A -85,B 0,C 180,E1 -23415.252,E2 -23415.252} C_VEL
LIN {X 0,Y 206.377,Z 375.048,A -85,B 0,C 180,E1 -23420.879,E2 -23420.879} C_VEL
LIN {X 0,Y 206.285,Z 375.413,A -85,B 0,C 180,E1 -23425.361,E2 -23425.361} C_VEL
LIN {X 0,Y 206.605,Z 376.19,A -85,B 0,C 180,E1 -23427.19,E2 -23427.19} C_VEL
LIN {X 0,Y 209.245,Z 381.704,A -85,B 0,C 180,E1 -23432.977,E2 -23432.977} C_VEL
LIN {X 0,Y 211.84,Z 387.285,A -85,B 0,C 180,E1 -23436.373,E2 -23436.373} C_VEL
LIN {X 0,Y 214.115,Z 392.585,A -85,B 0,C 180,E1 -23438.779,E2 -23438.779} C_VEL
LIN {X 0,Y 216.652,Z 398.822,A -85,B 0,C 180,E1 -23441.019,E2 -23441.019} C_VEL
LIN {X 0,Y 218.809,Z 405.059,A -85,B 0,C 180,E1 -23442.806,E2 -23442.806} C_VEL
LIN {X 0,Y 219.322,Z 406.63,A -85,B 0,C 180,E1 -23443.2,E2 -23443.2} C_VEL
LIN {X 0,Y 215.44,Z 440.72,A -85,B 0,C 180,E1 -23444.455,E2 -23444.455} C_VEL
LIN {X 0,Y 212.831,Z 453.919,A -85,B 0,C 180,E1 -23445.158,E2 -23445.158} C_VEL
LIN {X 0,Y 209.274,Z 466.847,A -85,B 0,C 180,E1 -23446.159,E2 -23446.159} C_VEL
LIN {X 0,Y 204.874,Z 479.283,A -85,B 0,C 180,E1 -23447.497,E2 -23447.497} C_VEL
LIN {X 0,Y 200.039,Z 490.6,A -85,B 0,C 180,E1 -23449.128,E2 -23449.128} C_VEL
LIN {X 0,Y 195.203,Z 500.303,A -85,B 0,C 180,E1 -23450.944,E2 -23450.944} C_VEL
LIN {X 0,Y 193.303,Z 503.849,A -85,B 0,C 180,E1 -23451.741,E2 -23451.741} C_VEL
LIN {X 0,Y 190.509,Z 508.09,A -85,B 0,C 180,E1 -23452.645,E2 -23452.645} C_VEL
LIN {X 0,Y 181.796,Z 517.173,A -85,B 0,C 180,E1 -23454.46,E2 -23454.46} C_VEL
LIN {X 0,Y 177.049,Z 521.865,A -85,B 0,C 180,E1 -23455.808,E2 -23455.808} C_VEL
LIN {X 0,Y 175.211,Z 523.981,A -85,B 0,C 180,E1 -23456.686,E2 -23456.686} C_VEL
LIN {X 0,Y 169.73,Z 530.632,A -85,B 0,C 180,E1 -23460.205,E2 -23460.205} C_VEL
LIN {X 0,Y 165.621,Z 535.253,A -85,B 0,C 180,E1 -23463.54,E2 -23463.54} C_VEL
LIN {X 0,Y 162.17,Z 538.852,A -85,B 0,C 180,E1 -23467.042,E2 -23467.042} C_VEL
LIN {X 0,Y 160.111,Z 540.741,A -85,B 0,C 180,E1 -23469.441,E2 -23469.441} C_VEL
LIN {X 0,Y 157.058,Z 543.273,A -85,B 0,C 180,E1 -23474.424,E2 -23474.424} C_VEL
LIN {X 0,Y 155.426,Z 544.317,A -85,B 0,C 180,E1 -23479.578,E2 -23479.578} C_VEL
LIN {X 0,Y 154.969,Z 544.245,A -85,B 0,C 180,E1 -23482.179,E2 -23482.179} C_VEL
LIN {X 0,Y 154.904,Z 542.928,A -85,B 0,C 180,E1 -23487.398,E2 -23487.398} C_VEL
LIN {X 0,Y 155.17,Z 541.682,A -85,B 0,C 180,E1 -23489.998,E2 -23489.998} C_VEL
LIN {X 0,Y 154.999,Z 538.773,A -85,B 0,C 180,E1 -23494.031,E2 -23494.031} C_VEL
LIN {X 0,Y 155.162,Z 534.986,A -85,B 0,C 180,E1 -23497.808,E2 -23497.808} C_VEL
LIN {X 0,Y 155.757,Z 529.888,A -85,B 0,C 180,E1 -23501.714,E2 -23501.714} C_VEL
LIN {X 0,Y 156.882,Z 523.399,A -85,B 0,C 180,E1 -23505.59,E2 -23505.59} C_VEL
LIN {X 0,Y 158.726,Z 515.264,A -85,B 0,C 180,E1 -23509.393,E2 -23509.393} C_VEL
LIN {X 0,Y 160.655,Z 506.934,A -85,B 0,C 180,E1 -23512.504,E2 -23512.504} C_VEL
LIN {X 0,Y 163.053,Z 496.768,A -85,B 0,C 180,E1 -23515.531,E2 -23515.531} C_VEL
LIN {X 0,Y 165.63,Z 485.297,A -85,B 0,C 180,E1 -23518.166,E2 -23518.166} C_VEL
LIN {X 0,Y 167.885,Z 474.143,A -85,B 0,C 180,E1 -23520.153,E2 -23520.153} C_VEL
LIN {X 0,Y 169.971,Z 461.793,A -85,B 0,C 180,E1 -23521.814,E2 -23521.814} C_VEL
LIN {X 0,Y 171.775,Z 448.351,A -85,B 0,C 180,E1 -23523.087,E2 -23523.087} C_VEL
LIN {X 0,Y 172.865,Z 435.229,A -85,B 0,C 180,E1 -23523.898,E2 -23523.898} C_VEL
LIN {X 0,Y 175.293,Z 393.525,A -85,B 0,C 180,E1 -23525.858,E2 -23525.858} C_VEL
LIN {X 0,Y 173.221,Z 373.721,A -85,B 0,C 180,E1 -23527.293,E2 -23527.293} C_VEL
LIN {X 0,Y 165.416,Z 351.465,A -85,B 0,C 180,E1 -23529.907,E2 -23529.907} C_VEL
LIN {X 0,Y 158.95,Z 336.033,A -85,B 0,C 180,E1 -23532.12,E2 -23532.12} C_VEL
LIN {X 0,Y 157.681,Z 332.907,A -85,B 0,C 180,E1 -23532.629,E2 -23532.629} C_VEL
LIN {X 0,Y 157.199,Z 330.904,A -85,B 0,C 180,E1 -23534.054,E2 -23534.054} C_VEL
LIN {X 0,Y 157.207,Z 330.904,A -85,B 0,C 180,E1 -23539.46,E2 -23539.46} C_VEL
LIN {X 0,Y 157.284,Z 330.894,A -85,B 0,C 180,E1 -23544.488,E2 -23544.488} C_VEL
LIN {X 0,Y 157.29,Z 330.871,A -85,B 0,C 180,E1 -23548.095,E2 -23548.095} C_VEL
LIN {X 0,Y 157.318,Z 330.887,A -85,B 0,C 180,E1 -23553.466,E2 -23553.466} C_VEL
LIN {X 0,Y 157.389,Z 330.872,A -85,B 0,C 180,E1 -23559.667,E2 -23559.667} C_VEL
LIN {X 0,Y 157.474,Z 330.869,A -85,B 0,C 180,E1 -23564.468,E2 -23564.468} C_VEL
LIN {X 0,Y 157.742,Z 330.827,A -85,B 0,C 180,E1 -23569.735,E2 -23569.735} C_VEL
LIN {X 0,Y 157.807,Z 330.826,A -85,B 0,C 180,E1 -23572.323,E2 -23572.323} C_VEL
LIN {X 0,Y 158.252,Z 330.755,A -85,B 0,C 180,E1 -23580.001,E2 -23580.001} C_VEL
LIN {X 0,Y 157.759,Z 330.826,A -85,B 0,C 180,E1 -23587.681,E2 -23587.681} C_VEL
LIN {X 0,Y 157.632,Z 330.824,A -85,B 0,C 180,E1 -23591.237,E2 -23591.237} C_VEL
LIN {X 0,Y 157.45,Z 330.863,A -85,B 0,C 180,E1 -23595.535,E2 -23595.535} C_VEL
LIN {X 0,Y 157.364,Z 330.875,A -85,B 0,C 180,E1 -23600.934,E2 -23600.934} C_VEL
LIN {X 0,Y 157.306,Z 330.866,A -85,B 0,C 180,E1 -23606.682,E2 -23606.682} C_VEL
LIN {X 0,Y 157.265,Z 330.895,A -85,B 0,C 180,E1 -23612.431,E2 -23612.431} C_VEL
LIN {X 0,Y 157.265,Z 330.888,A -85,B 0,C 180,E1 -23616.451,E2 -23616.451} C_VEL
LIN {X 0,Y 157.191,Z 330.891,A -85,B 0,C 180,E1 -23622.118,E2 -23622.118} C_VEL
LIN {X 0,Y 157.189,Z 330.903,A -85,B 0,C 180,E1 -23627.885,E2 -23627.885} C_VEL
LIN {X 0,Y 157.258,Z 330.881,A -85,B 0,C 180,E1 -23633.557,E2 -23633.557} C_VEL
LIN {X 0,Y 157.283,Z 330.892,A -85,B 0,C 180,E1 -23638.104,E2 -23638.104} C_VEL
LIN {X 0,Y 157.31,Z 330.891,A -85,B 0,C 180,E1 -23643.466,E2 -23643.466} C_VEL
LIN {X 0,Y 157.379,Z 330.879,A -85,B 0,C 180,E1 -23649.686,E2 -23649.686} C_VEL
LIN {X 0,Y 157.426,Z 330.873,A -85,B 0,C 180,E1 -23654.465,E2 -23654.465} C_VEL
LIN {X 0,Y 157.69,Z 330.843,A -85,B 0,C 180,E1 -23659.732,E2 -23659.732} C_VEL
LIN {X 0,Y 157.761,Z 330.835,A -85,B 0,C 180,E1 -23662.321,E2 -23662.321} C_VEL
LIN {X 0,Y 158.234,Z 330.777,A -85,B 0,C 180,E1 -23670.001,E2 -23670.001} C_VEL
LIN {X 0,Y 157.694,Z 330.845,A -85,B 0,C 180,E1 -23675.035,E2 -23675.035} C_VEL
LIN {X 0,Y 158.672,Z 333.634,A -85,B 0,C 180,E1 -23675.442,E2 -23675.442} C_VEL
LIN {X 0,Y 163.616,Z 343.262,A -85,B 0,C 180,E1 -23677.021,E2 -23677.021} C_VEL
LIN {X 0,Y 173.16,Z 365.12,A -85,B 0,C 180,E1 -23679.97,E2 -23679.97} C_VEL
LIN {X 0,Y 176.187,Z 373.714,A -85,B 0,C 180,E1 -23680.928,E2 -23680.928} C_VEL
LIN {X 0,Y 172.577,Z 430.341,A -85,B 0,C 180,E1 -23683.605,E2 -23683.605} C_VEL
LIN {X 0,Y 171.144,Z 444.091,A -85,B 0,C 180,E1 -23684.721,E2 -23684.721} C_VEL
LIN {X 0,Y 169.383,Z 457.015,A -85,B 0,C 180,E1 -23686.266,E2 -23686.266} C_VEL
LIN {X 0,Y 167.4,Z 468.173,A -85,B 0,C 180,E1 -23688.038,E2 -23688.038} C_VEL
LIN {X 0,Y 165.005,Z 479.884,A -85,B 0,C 180,E1 -23690.438,E2 -23690.438} C_VEL
LIN {X 0,Y 162.669,Z 490.325,A -85,B 0,C 180,E1 -23693.189,E2 -23693.189} C_VEL
LIN {X 0,Y 160.385,Z 499.805,A -85,B 0,C 180,E1 -23696.336,E2 -23696.336} C_VEL
LIN {X 0,Y 158.373,Z 508.226,A -85,B 0,C 180,E1 -23699.838,E2 -23699.838} C_VEL
LIN {X 0,Y 156.837,Z 514.874,A -85,B 0,C 180,E1 -23703.295,E2 -23703.295} C_VEL
LIN {X 0,Y 155.644,Z 521.295,A -85,B 0,C 180,E1 -23707.559,E2 -23707.559} C_VEL
LIN {X 0,Y 154.738,Z 525.59,A -85,B 0,C 180,E1 -23711.22,E2 -23711.22} C_VEL
LIN {X 0,Y 154.334,Z 529.061,A -85,B 0,C 180,E1 -23715.104,E2 -23715.104} C_VEL
LIN {X 0,Y 154.327,Z 530.342,A -85,B 0,C 180,E1 -23716.913,E2 -23716.913} C_VEL
LIN {X 0,Y 154.599,Z 532.302,A -85,B 0,C 180,E1 -23720.609,E2 -23720.609} C_VEL
LIN {X 0,Y 155.378,Z 533.474,A -85,B 0,C 180,E1 -23724.507,E2 -23724.507} C_VEL
LIN {X 0,Y 156.695,Z 533.77,A -85,B 0,C 180,E1 -23728.452,E2 -23728.452} C_VEL
LIN {X 0,Y 158.665,Z 533.141,A -85,B 0,C 180,E1 -23732.364,E2 -23732.364} C_VEL
LIN {X 0,Y 161.848,Z 531.124,A -85,B 0,C 180,E1 -23736.994,E2 -23736.994} C_VEL
LIN {X 0,Y 166.14,Z 527.539,A -85,B 0,C 180,E1 -23741.502,E2 -23741.502} C_VEL
LIN {X 0,Y 171.38,Z 522.336,A -85,B 0,C 180,E1 -23745.755,E2 -23745.755} C_VEL
LIN {X 0,Y 176.084,Z 516.912,A -85,B 0,C 180,E1 -23748.947,E2 -23748.947} C_VEL
LIN {X 0,Y 181.919,Z 509.34,A -85,B 0,C 180,E1 -23752.23,E2 -23752.23} C_VEL
LIN {X 0,Y 187.359,Z 501.283,A -85,B 0,C 180,E1 -23754.888,E2 -23754.888} C_VEL
LIN {X 0,Y 192.63,Z 492.473,A -85,B 0,C 180,E1 -23757.124,E2 -23757.124} C_VEL
LIN {X 0,Y 198.011,Z 481.918,A -85,B 0,C 180,E1 -23759.192,E2 -23759.192} C_VEL
LIN {X 0,Y 203.166,Z 469.756,A -85,B 0,C 180,E1 -23760.976,E2 -23760.976} C_VEL
LIN {X 0,Y 207.28,Z 457.452,A -85,B 0,C 180,E1 -23762.344,E2 -23762.344} C_VEL
LIN {X 0,Y 210.705,Z 443.973,A -85,B 0,C 180,E1 -23763.437,E2 -23763.437} C_VEL
LIN {X 0,Y 213.055,Z 431.079,A -85,B 0,C 180,E1 -23764.114,E2 -23764.114} C_VEL
LIN {X 0,Y 216.39,Z 402.612,A -85,B 0,C 180,E1 -23765.15,E2 -23765.15} C_VEL
LIN {X 0,Y 213.403,Z 395.598,A -85,B 0,C 180,E1 -23767.759,E2 -23767.759} C_VEL
LIN {X 0,Y 211.456,Z 392.236,A -85,B 0,C 180,E1 -23769.654,E2 -23769.654} C_VEL
LIN {X 0,Y 208.995,Z 387.964,A -85,B 0,C 180,E1 -23772.542,E2 -23772.542} C_VEL
LIN {X 0,Y 207.091,Z 384.571,A -85,B 0,C 180,E1 -23775.553,E2 -23775.553} C_VEL
LIN {X 0,Y 205.207,Z 382.027,A -85,B 0,C 180,E1 -23781.003,E2 -23781.003} C_VEL
LIN {X 0,Y 205.152,Z 382.487,A -85,B 0,C 180,E1 -23785.511,E2 -23785.511} C_VEL
LIN {X 0,Y 205.398,Z 383.275,A -85,B 0,C 180,E1 -23787.085,E2 -23787.085} C_VEL
LIN {X 0,Y 207.708,Z 388.443,A -85,B 0,C 180,E1 -23792.497,E2 -23792.497} C_VEL
LIN {X 0,Y 210.006,Z 393.908,A -85,B 0,C 180,E1 -23795.785,E2 -23795.785} C_VEL
LIN {X 0,Y 211.809,Z 398.319,A -85,B 0,C 180,E1 -23797.831,E2 -23797.831} C_VEL
LIN {X 0,Y 213.99,Z 404.125,A -85,B 0,C 180,E1 -23799.982,E2 -23799.982} C_VEL
LIN {X 0,Y 215.776,Z 409.648,A -85,B 0,C 180,E1 -23801.619,E2 -23801.619} C_VEL
LIN {X 0,Y 212.002,Z 440.875,A -85,B 0,C 180,E1 -23802.789,E2 -23802.789} C_VEL
LIN {X 0,Y 209.387,Z 453.596,A -85,B 0,C 180,E1 -23803.46,E2 -23803.46} C_VEL
LIN {X 0,Y 206.229,Z 464.931,A -85,B 0,C 180,E1 -23804.302,E2 -23804.302} C_VEL
LIN {X 0,Y 201.91,Z 477.073,A -85,B 0,C 180,E1 -23805.531,E2 -23805.531} C_VEL
LIN {X 0,Y 197.197,Z 488.04,A -85,B 0,C 180,E1 -23807.03,E2 -23807.03} C_VEL
LIN {X 0,Y 191.48,Z 499.162,A -85,B 0,C 180,E1 -23808.997,E2 -23808.997} C_VEL
LIN {X 0,Y 185.72,Z 508.93,A -85,B 0,C 180,E1 -23811.361,E2 -23811.361} C_VEL
LIN {X 0,Y 179.79,Z 517.706,A -85,B 0,C 180,E1 -23814.1,E2 -23814.1} C_VEL
LIN {X 0,Y 175.211,Z 523.981,A -85,B 0,C 180,E1 -23816.686,E2 -23816.686} C_VEL
LIN {X 0,Y 172.301,Z 527.071,A -85,B 0,C 180,E1 -23818.046,E2 -23818.046} C_VEL
LIN {X 0,Y 166.037,Z 531.674,A -85,B 0,C 180,E1 -23820.136,E2 -23820.136} C_VEL
LIN {X 0,Y 159.918,Z 535.587,A -85,B 0,C 180,E1 -23822.501,E2 -23822.501} C_VEL
LIN {X 0,Y 157.312,Z 537.527,A -85,B 0,C 180,E1 -23824.272,E2 -23824.272} C_VEL
LIN {X 0,Y 153.483,Z 540.815,A -85,B 0,C 180,E1 -23828.51,E2 -23828.51} C_VEL
LIN {X 0,Y 150.194,Z 543.189,A -85,B 0,C 180,E1 -23833.693,E2 -23833.693} C_VEL
LIN {X 0,Y 149.169,Z 543.81,A -85,B 0,C 180,E1 -23836.373,E2 -23836.373} C_VEL
LIN {X 0,Y 147.936,Z 543.861,A -85,B 0,C 180,E1 -23841.805,E2 -23841.805} C_VEL
LIN {X 0,Y 147.823,Z 542.413,A -85,B 0,C 180,E1 -23847.273,E2 -23847.273} C_VEL
LIN {X 0,Y 148.108,Z 541.075,A -85,B 0,C 180,E1 -23849.998,E2 -23849.998} C_VEL
LIN {X 0,Y 147.932,Z 538.281,A -85,B 0,C 180,E1 -23853.915,E2 -23853.915} C_VEL
LIN {X 0,Y 148.138,Z 534.081,A -85,B 0,C 180,E1 -23858.181,E2 -23858.181} C_VEL
LIN {X 0,Y 148.949,Z 527.748,A -85,B 0,C 180,E1 -23862.95,E2 -23862.95} C_VEL
LIN {X 0,Y 150.327,Z 520.805,A -85,B 0,C 180,E1 -23866.988,E2 -23866.988} C_VEL
LIN {X 0,Y 152.005,Z 513.698,A -85,B 0,C 180,E1 -23870.288,E2 -23870.288} C_VEL
LIN {X 0,Y 154.096,Z 505.097,A -85,B 0,C 180,E1 -23873.518,E2 -23873.518} C_VEL
LIN {X 0,Y 156.612,Z 494.463,A -85,B 0,C 180,E1 -23876.662,E2 -23876.662} C_VEL
LIN {X 0,Y 159.033,Z 484.021,A -85,B 0,C 180,E1 -23879.083,E2 -23879.083} C_VEL
LIN {X 0,Y 161.433,Z 472.663,A -85,B 0,C 180,E1 -23881.128,E2 -23881.128} C_VEL
LIN {X 0,Y 163.593,Z 459.878,A -85,B 0,C 180,E1 -23882.843,E2 -23882.843} C_VEL
LIN {X 0,Y 165.356,Z 446.736,A -85,B 0,C 180,E1 -23884.088,E2 -23884.088} C_VEL
LIN {X 0,Y 166.518,Z 431.194,A -85,B 0,C 180,E1 -23885.009,E2 -23885.009} C_VEL
LIN {X 0,Y 168.824,Z 394.348,A -85,B 0,C 180,E1 -23886.798,E2 -23886.798} C_VEL
LIN {X 0,Y 166.973,Z 375.973,A -85,B 0,C 180,E1 -23888.166,E2 -23888.166} C_VEL
LIN {X 0,Y 159.191,Z 353.616,A -85,B 0,C 180,E1 -23890.945,E2 -23890.945} C_VEL
LIN {X 0,Y 153.343,Z 339.551,A -85,B 0,C 180,E1 -23893.061,E2 -23893.061} C_VEL
LIN {X 0,Y 150.294,Z 332.593,A -85,B 0,C 180,E1 -23894.271,E2 -23894.271} C_VEL
LIN {X 0,Y 150.122,Z 331.787,A -85,B 0,C 180,E1 -23894.891,E2 -23894.891} C_VEL
LIN {X 0,Y 150.152,Z 331.784,A -85,B 0,C 180,E1 -23899.059,E2 -23899.059} C_VEL
LIN {X 0,Y 150.211,Z 331.773,A -85,B 0,C 180,E1 -23902.689,E2 -23902.689} C_VEL
LIN {X 0,Y 150.213,Z 331.76,A -85,B 0,C 180,E1 -23907.366,E2 -23907.366} C_VEL
LIN {X 0,Y 150.24,Z 331.763,A -85,B 0,C 180,E1 -23912.717,E2 -23912.717} C_VEL
LIN {X 0,Y 150.347,Z 331.749,A -85,B 0,C 180,E1 -23919.208,E2 -23919.208} C_VEL
LIN {X 0,Y 150.379,Z 331.754,A -85,B 0,C 180,E1 -23923.716,E2 -23923.716} C_VEL
LIN {X 0,Y 150.66,Z 331.706,A -85,B 0,C 180,E1 -23929.247,E2 -23929.247} C_VEL
LIN {X 0,Y 150.744,Z 331.707,A -85,B 0,C 180,E1 -23931.961,E2 -23931.961} C_VEL
LIN {X 0,Y 151.213,Z 331.631,A -85,B 0,C 180,E1 -23940.001,E2 -23940.001} C_VEL
LIN {X 0,Y 150.697,Z 331.703,A -85,B 0,C 180,E1 -23948.043,E2 -23948.043} C_VEL
LIN {X 0,Y 150.573,Z 331.702,A -85,B 0,C 180,E1 -23951.437,E2 -23951.437} C_VEL
LIN {X 0,Y 150.358,Z 331.749,A -85,B 0,C 180,E1 -23956.288,E2 -23956.288} C_VEL
LIN {X 0,Y 150.346,Z 331.749,A -85,B 0,C 180,E1 -23960.792,E2 -23960.792} C_VEL
LIN {X 0,Y 150.235,Z 331.751,A -85,B 0,C 180,E1 -23967.279,E2 -23967.279} C_VEL
LIN {X 0,Y 150.206,Z 331.776,A -85,B 0,C 180,E1 -23972.63,E2 -23972.63} C_VEL
LIN {X 0,Y 150.17,Z 331.766,A -85,B 0,C 180,E1 -23977.475,E2 -23977.475} C_VEL
LIN {X 0,Y 150.134,Z 331.765,A -85,B 0,C 180,E1 -23981.5,E2 -23981.5} C_VEL
LIN {X 0,Y 150.125,Z 331.784,A -85,B 0,C 180,E1 -23985.398,E2 -23985.398} C_VEL
LIN {X 0,Y 150.137,Z 331.779,A -85,B 0,C 180,E1 -23989.056,E2 -23989.056} C_VEL
LIN {X 0,Y 150.175,Z 331.76,A -85,B 0,C 180,E1 -23992.712,E2 -23992.712} C_VEL
LIN {X 0,Y 150.208,Z 331.775,A -85,B 0,C 180,E1 -23997.374,E2 -23997.374} C_VEL
LIN {X 0,Y 150.239,Z 331.77,A -85,B 0,C 180,E1 -24002.725,E2 -24002.725} C_VEL
LIN {X 0,Y 150.34,Z 331.756,A -85,B 0,C 180,E1 -24009.222,E2 -24009.222} C_VEL
LIN {X 0,Y 150.333,Z 331.756,A -85,B 0,C 180,E1 -24013.712,E2 -24013.712} C_VEL
LIN {X 0,Y 150.611,Z 331.723,A -85,B 0,C 180,E1 -24019.244,E2 -24019.244} C_VEL
LIN {X 0,Y 150.684,Z 331.715,A -85,B 0,C 180,E1 -24021.958,E2 -24021.958} C_VEL
LIN {X 0,Y 151.194,Z 331.654,A -85,B 0,C 180,E1 -24030.002,E2 -24030.002} C_VEL
LIN {X 0,Y 150.725,Z 331.713,A -85,B 0,C 180,E1 -24033.594,E2 -24033.594} C_VEL
LIN {X 0,Y 151.684,Z 334.524,A -85,B 0,C 180,E1 -24034.016,E2 -24034.016} C_VEL
LIN {X 0,Y 158.001,Z 346.838,A -85,B 0,C 180,E1 -24036.144,E2 -24036.144} C_VEL
LIN {X 0,Y 167.118,Z 367.862,A -85,B 0,C 180,E1 -24039.137,E2 -24039.137} C_VEL
LIN {X 0,Y 169.761,Z 375.332,A -85,B 0,C 180,E1 -24040.011,E2 -24040.011} C_VEL
LIN {X 0,Y 165.968,Z 430.804,A -85,B 0,C 180,E1 -24042.727,E2 -24042.727} C_VEL
LIN {X 0,Y 164.56,Z 443.872,A -85,B 0,C 180,E1 -24043.82,E2 -24043.82} C_VEL
LIN {X 0,Y 162.702,Z 457.078,A -85,B 0,C 180,E1 -24045.437,E2 -24045.437} C_VEL
LIN {X 0,Y 160.381,Z 469.66,A -85,B 0,C 180,E1 -24047.535,E2 -24047.535} C_VEL
LIN {X 0,Y 158.124,Z 480.217,A -85,B 0,C 180,E1 -24049.811,E2 -24049.811} C_VEL
LIN {X 0,Y 155.811,Z 490.233,A -85,B 0,C 180,E1 -24052.546,E2 -24052.546} C_VEL
LIN {X 0,Y 153.423,Z 499.801,A -85,B 0,C 180,E1 -24055.834,E2 -24055.834} C_VEL
LIN {X 0,Y 151.305,Z 508.412,A -85,B 0,C 180,E1 -24059.557,E2 -24059.557} C_VEL
LIN {X 0,Y 149.712,Z 515.336,A -85,B 0,C 180,E1 -24063.332,E2 -24063.332} C_VEL
LIN {X 0,Y 148.764,Z 520.13,A -85,B 0,C 180,E1 -24066.569,E2 -24066.569} C_VEL
LIN {X 0,Y 147.765,Z 524.776,A -85,B 0,C 180,E1 -24070.447,E2 -24070.447} C_VEL
LIN {X 0,Y 147.284,Z 528.325,A -85,B 0,C 180,E1 -24074.293,E2 -24074.293} C_VEL
LIN {X 0,Y 147.382,Z 531.839,A -85,B 0,C 180,E1 -24079.729,E2 -24079.729} C_VEL
LIN {X 0,Y 148.063,Z 533.396,A -85,B 0,C 180,E1 -24083.799,E2 -24083.799} C_VEL
LIN {X 0,Y 149.717,Z 534.081,A -85,B 0,C 180,E1 -24088.911,E2 -24088.911} C_VEL
LIN {X 0,Y 151.426,Z 533.767,A -85,B 0,C 180,E1 -24092.346,E2 -24092.346} C_VEL
LIN {X 0,Y 153.818,Z 532.632,A -85,B 0,C 180,E1 -24096.04,E2 -24096.04} C_VEL
LIN {X 0,Y 157.104,Z 530.473,A -85,B 0,C 180,E1 -24099.959,E2 -24099.959} C_VEL
LIN {X 0,Y 161.09,Z 527.277,A -85,B 0,C 180,E1 -24103.705,E2 -24103.705} C_VEL
LIN {X 0,Y 166.577,Z 522.141,A -85,B 0,C 180,E1 -24107.821,E2 -24107.821} C_VEL
LIN {X 0,Y 172.095,Z 516.107,A -85,B 0,C 180,E1 -24111.257,E2 -24111.257} C_VEL
LIN {X 0,Y 177.237,Z 509.793,A -85,B 0,C 180,E1 -24113.986,E2 -24113.986} C_VEL
LIN {X 0,Y 183.041,Z 501.699,A -85,B 0,C 180,E1 -24116.664,E2 -24116.664} C_VEL
LIN {X 0,Y 189.263,Z 491.677,A -85,B 0,C 180,E1 -24119.174,E2 -24119.174} C_VEL
LIN {X 0,Y 195.142,Z 480.354,A -85,B 0,C 180,E1 -24121.29,E2 -24121.29} C_VEL
LIN {X 0,Y 200.132,Z 468.937,A -85,B 0,C 180,E1 -24122.893,E2 -24122.893} C_VEL
LIN {X 0,Y 204.367,Z 456.561,A -85,B 0,C 180,E1 -24124.213,E2 -24124.213} C_VEL
LIN {X 0,Y 207.5,Z 444.648,A -85,B 0,C 180,E1 -24125.156,E2 -24125.156} C_VEL
LIN {X 0,Y 210.026,Z 431.271,A -85,B 0,C 180,E1 -24125.855,E2 -24125.855} C_VEL
LIN {X 0,Y 213.047,Z 406.251,A -85,B 0,C 180,E1 -24126.772,E2 -24126.772} C_VEL
LIN {X 0,Y 210.984,Z 401.07,A -85,B 0,C 180,E1 -24128.84,E2 -24128.84} C_VEL
LIN {X 0,Y 208.921,Z 397.668,A -85,B 0,C 180,E1 -24130.994,E2 -24130.994} C_VEL
LIN {X 0,Y 207.334,Z 394.516,A -85,B 0,C 180,E1 -24133.153,E2 -24133.153} C_VEL
LIN {X 0,Y 205.758,Z 391.461,A -85,B 0,C 180,E1 -24135.858,E2 -24135.858} C_VEL
LIN {X 0,Y 204.035,Z 389.03,A -85,B 0,C 180,E1 -24141.13,E2 -24141.13} C_VEL
LIN {X 0,Y 203.963,Z 389.426,A -85,B 0,C 180,E1 -24145.225,E2 -24145.225} C_VEL
LIN {X 0,Y 204.181,Z 390.261,A -85,B 0,C 180,E1 -24146.839,E2 -24146.839} C_VEL
LIN {X 0,Y 206.098,Z 395.016,A -85,B 0,C 180,E1 -24151.868,E2 -24151.868} C_VEL
LIN {X 0,Y 208.084,Z 400.187,A -85,B 0,C 180,E1 -24155.041,E2 -24155.041} C_VEL
LIN {X 0,Y 209.77,Z 404.607,A -85,B 0,C 180,E1 -24157.089,E2 -24157.089} C_VEL
LIN {X 0,Y 211.843,Z 410.842,A -85,B 0,C 180,E1 -24159.374,E2 -24159.374} C_VEL
LIN {X 0,Y 212.48,Z 412.837,A -85,B 0,C 180,E1 -24159.997,E2 -24159.997} C_VEL
LIN {X 0,Y 209.037,Z 440.277,A -85,B 0,C 180,E1 -24161.018,E2 -24161.018} C_VEL
LIN {X 0,Y 206.054,Z 454.154,A -85,B 0,C 180,E1 -24161.745,E2 -24161.745} C_VEL
LIN {X 0,Y 202.136,Z 467.048,A -85,B 0,C 180,E1 -24162.735,E2 -24162.735} C_VEL
LIN {X 0,Y 197.04,Z 480.104,A -85,B 0,C 180,E1 -24164.124,E2 -24164.124} C_VEL
LIN {X 0,Y 191.56,Z 491.549,A -85,B 0,C 180,E1 -24165.806,E2 -24165.806} C_VEL
LIN {X 0,Y 185.737,Z 501.904,A -85,B 0,C 180,E1 -24167.805,E2 -24167.805} C_VEL
LIN {X 0,Y 180.33,Z 510.394,A -85,B 0,C 180,E1 -24169.979,E2 -24169.979} C_VEL
LIN {X 0,Y 174.154,Z 518.8,A -85,B 0,C 180,E1 -24172.746,E2 -24172.746} C_VEL
LIN {X 0,Y 167.836,Z 526.603,A -85,B 0,C 180,E1 -24176.299,E2 -24176.299} C_VEL
LIN {X 0,Y 161.844,Z 533.06,A -85,B 0,C 180,E1 -24180.283,E2 -24180.283} C_VEL
LIN {X 0,Y 157.312,Z 537.527,A -85,B 0,C 180,E1 -24184.272,E2 -24184.272} C_VEL
LIN {X 0,Y 154.831,Z 539.254,A -85,B 0,C 180,E1 -24186.143,E2 -24186.143} C_VEL
LIN {X 0,Y 149.341,Z 541.509,A -85,B 0,C 180,E1 -24189.146,E2 -24189.146} C_VEL
LIN {X 0,Y 144.307,Z 542.942,A -85,B 0,C 180,E1 -24192.426,E2 -24192.426} C_VEL
LIN {X 0,Y 142.612,Z 543.396,A -85,B 0,C 180,E1 -24194.67,E2 -24194.67} C_VEL
LIN {X 0,Y 141.423,Z 543.712,A -85,B 0,C 180,E1 -24198.533,E2 -24198.533} C_VEL
LIN {X 0,Y 140.654,Z 542.863,A -85,B 0,C 180,E1 -24204.263,E2 -24204.263} C_VEL
LIN {X 0,Y 140.755,Z 541.836,A -85,B 0,C 180,E1 -24207.136,E2 -24207.136} C_VEL
LIN {X 0,Y 141.045,Z 540.391,A -85,B 0,C 180,E1 -24209.998,E2 -24209.998} C_VEL
LIN {X 0,Y 140.867,Z 537.74,A -85,B 0,C 180,E1 -24213.789,E2 -24213.789} C_VEL
LIN {X 0,Y 141.091,Z 533.095,A -85,B 0,C 180,E1 -24218.592,E2 -24218.592} C_VEL
LIN {X 0,Y 141.822,Z 527.625,A -85,B 0,C 180,E1 -24222.883,E2 -24222.883} C_VEL
LIN {X 0,Y 143.203,Z 520.712,A -85,B 0,C 180,E1 -24227.123,E2 -24227.123} C_VEL
LIN {X 0,Y 144.935,Z 513.644,A -85,B 0,C 180,E1 -24230.581,E2 -24230.581} C_VEL
LIN {X 0,Y 147.078,Z 505.096,A -85,B 0,C 180,E1 -24233.962,E2 -24233.962} C_VEL
LIN {X 0,Y 149.53,Z 495.262,A -85,B 0,C 180,E1 -24237.04,E2 -24237.04} C_VEL
LIN {X 0,Y 152.189,Z 484.155,A -85,B 0,C 180,E1 -24239.762,E2 -24239.762} C_VEL
LIN {X 0,Y 154.634,Z 472.903,A -85,B 0,C 180,E1 -24241.892,E2 -24241.892} C_VEL
LIN {X 0,Y 156.88,Z 460.306,A -85,B 0,C 180,E1 -24243.666,E2 -24243.666} C_VEL
LIN {X 0,Y 158.777,Z 446.57,A -85,B 0,C 180,E1 -24245.03,E2 -24245.03} C_VEL
LIN {X 0,Y 159.941,Z 431.819,A -85,B 0,C 180,E1 -24245.946,E2 -24245.946} C_VEL
LIN {X 0,Y 162.343,Z 394.795,A -85,B 0,C 180,E1 -24247.809,E2 -24247.809} C_VEL
LIN {X 0,Y 160.6,Z 377.699,A -85,B 0,C 180,E1 -24249.16,E2 -24249.16} C_VEL
LIN {X 0,Y 153.108,Z 355.994,A -85,B 0,C 180,E1 -24252.009,E2 -24252.009} C_VEL
LIN {X 0,Y 146.481,Z 340.129,A -85,B 0,C 180,E1 -24254.55,E2 -24254.55} C_VEL
LIN {X 0,Y 144.21,Z 335.697,A -85,B 0,C 180,E1 -24255.406,E2 -24255.406} C_VEL
LIN {X 0,Y 143.143,Z 333.178,A -85,B 0,C 180,E1 -24255.848,E2 -24255.848} C_VEL
LIN {X 0,Y 143.047,Z 332.663,A -85,B 0,C 180,E1 -24256.055,E2 -24256.055} C_VEL
LIN {X 0,Y 143.103,Z 332.661,A -85,B 0,C 180,E1 -24261.79,E2 -24261.79} C_VEL
LIN {X 0,Y 143.181,Z 332.634,A -85,B 0,C 180,E1 -24267.321,E2 -24267.321} C_VEL
LIN {X 0,Y 143.186,Z 332.636,A -85,B 0,C 180,E1 -24272.062,E2 -24272.062} C_VEL
LIN {X 0,Y 143.273,Z 332.632,A -85,B 0,C 180,E1 -24278.745,E2 -24278.745} C_VEL
LIN {X 0,Y 143.312,Z 332.634,A -85,B 0,C 180,E1 -24282.889,E2 -24282.889} C_VEL
LIN {X 0,Y 143.59,Z 332.584,A -85,B 0,C 180,E1 -24288.71,E2 -24288.71} C_VEL
LIN {X 0,Y 143.665,Z 332.587,A -85,B 0,C 180,E1 -24291.562,E2 -24291.562} C_VEL
LIN {X 0,Y 144.171,Z 332.507,A -85,B 0,C 180,E1 -24300.001,E2 -24300.001} C_VEL
LIN {X 0,Y 143.619,Z 332.582,A -85,B 0,C 180,E1 -24308.443,E2 -24308.443} C_VEL
LIN {X 0,Y 143.501,Z 332.582,A -85,B 0,C 180,E1 -24311.629,E2 -24311.629} C_VEL
LIN {X 0,Y 143.297,Z 332.63,A -85,B 0,C 180,E1 -24317.115,E2 -24317.115} C_VEL
LIN {X 0,Y 143.271,Z 332.629,A -85,B 0,C 180,E1 -24321.253,E2 -24321.253} C_VEL
LIN {X 0,Y 143.179,Z 332.633,A -85,B 0,C 180,E1 -24327.933,E2 -24327.933} C_VEL
LIN {X 0,Y 143.136,Z 332.654,A -85,B 0,C 180,E1 -24333.419,E2 -24333.419} C_VEL
LIN {X 0,Y 143.053,Z 332.639,A -85,B 0,C 180,E1 -24339.694,E2 -24339.694} C_VEL
LIN {X 0,Y 143.032,Z 332.661,A -85,B 0,C 180,E1 -24343.465,E2 -24343.465} C_VEL
LIN {X 0,Y 143.037,Z 332.666,A -85,B 0,C 180,E1 -24347.479,E2 -24347.479} C_VEL
LIN {X 0,Y 143.071,Z 332.645,A -85,B 0,C 180,E1 -24351.811,E2 -24351.811} C_VEL
LIN {X 0,Y 143.175,Z 332.65,A -85,B 0,C 180,E1 -24357.322,E2 -24357.322} C_VEL
LIN {X 0,Y 143.183,Z 332.649,A -85,B 0,C 180,E1 -24362.071,E2 -24362.071} C_VEL
LIN {X 0,Y 143.268,Z 332.637,A -85,B 0,C 180,E1 -24368.758,E2 -24368.758} C_VEL
LIN {X 0,Y 143.271,Z 332.636,A -85,B 0,C 180,E1 -24372.885,E2 -24372.885} C_VEL
LIN {X 0,Y 143.537,Z 332.604,A -85,B 0,C 180,E1 -24378.707,E2 -24378.707} C_VEL
LIN {X 0,Y 143.61,Z 332.594,A -85,B 0,C 180,E1 -24381.559,E2 -24381.559} C_VEL
LIN {X 0,Y 144.152,Z 332.531,A -85,B 0,C 180,E1 -24390.002,E2 -24390.002} C_VEL
LIN {X 0,Y 143.851,Z 332.569,A -85,B 0,C 180,E1 -24392.014,E2 -24392.014} C_VEL
LIN {X 0,Y 144.813,Z 335.423,A -85,B 0,C 180,E1 -24392.479,E2 -24392.479} C_VEL
LIN {X 0,Y 152.502,Z 350.708,A -85,B 0,C 180,E1 -24395.29,E2 -24395.29} C_VEL
LIN {X 0,Y 161.28,Z 371.183,A -85,B 0,C 180,E1 -24398.314,E2 -24398.314} C_VEL
LIN {X 0,Y 163.26,Z 376.785,A -85,B 0,C 180,E1 -24399.011,E2 -24399.011} C_VEL
LIN {X 0,Y 159.465,Z 430.703,A -85,B 0,C 180,E1 -24401.739,E2 -24401.739} C_VEL
LIN {X 0,Y 157.909,Z 444.576,A -85,B 0,C 180,E1 -24402.941,E2 -24402.941} C_VEL
LIN {X 0,Y 156.109,Z 456.909,A -85,B 0,C 180,E1 -24404.504,E2 -24404.504} C_VEL
LIN {X 0,Y 153.799,Z 469.1,A -85,B 0,C 180,E1 -24406.586,E2 -24406.586} C_VEL
LIN {X 0,Y 151.438,Z 479.844,A -85,B 0,C 180,E1 -24408.959,E2 -24408.959} C_VEL
LIN {X 0,Y 149.046,Z 489.839,A -85,B 0,C 180,E1 -24411.748,E2 -24411.748} C_VEL
LIN {X 0,Y 146.639,Z 499.176,A -85,B 0,C 180,E1 -24415.036,E2 -24415.036} C_VEL
LIN {X 0,Y 144.278,Z 508.375,A -85,B 0,C 180,E1 -24419.153,E2 -24419.153} C_VEL
LIN {X 0,Y 142.428,Z 516.393,A -85,B 0,C 180,E1 -24423.806,E2 -24423.806} C_VEL
LIN {X 0,Y 141.414,Z 521.222,A -85,B 0,C 180,E1 -24427.327,E2 -24427.327} C_VEL
LIN {X 0,Y 140.493,Z 525.659,A -85,B 0,C 180,E1 -24431.377,E2 -24431.377} C_VEL
LIN {X 0,Y 140.142,Z 529.055,A -85,B 0,C 180,E1 -24435.404,E2 -24435.404} C_VEL
LIN {X 0,Y 140.241,Z 531.515,A -85,B 0,C 180,E1 -24439.346,E2 -24439.346} C_VEL
LIN {X 0,Y 140.808,Z 533.188,A -85,B 0,C 180,E1 -24443.205,E2 -24443.205} C_VEL
LIN {X 0,Y 141.947,Z 534.192,A -85,B 0,C 180,E1 -24447.322,E2 -24447.322} C_VEL
LIN {X 0,Y 143.779,Z 534.345,A -85,B 0,C 180,E1 -24451.627,E2 -24451.627} C_VEL
LIN {X 0,Y 146.359,Z 533.565,A -85,B 0,C 180,E1 -24455.836,E2 -24455.836} C_VEL
LIN {X 0,Y 150.541,Z 531.255,A -85,B 0,C 180,E1 -24460.925,E2 -24460.925} C_VEL
LIN {X 0,Y 155.753,Z 527.445,A -85,B 0,C 180,E1 -24465.63,E2 -24465.63} C_VEL
LIN {X 0,Y 161.953,Z 521.999,A -85,B 0,C 180,E1 -24470.003,E2 -24470.003} C_VEL
LIN {X 0,Y 168.317,Z 515.437,A -85,B 0,C 180,E1 -24473.633,E2 -24473.633} C_VEL
LIN {X 0,Y 173.987,Z 508.68,A -85,B 0,C 180,E1 -24476.43,E2 -24476.43} C_VEL
LIN {X 0,Y 180.464,Z 499.927,A -85,B 0,C 180,E1 -24479.163,E2 -24479.163} C_VEL
LIN {X 0,Y 186.351,Z 490.647,A -85,B 0,C 180,E1 -24481.35,E2 -24481.35} C_VEL
LIN {X 0,Y 191.82,Z 480.536,A -85,B 0,C 180,E1 -24483.182,E2 -24483.182} C_VEL
LIN {X 0,Y 196.877,Z 469.406,A -85,B 0,C 180,E1 -24484.711,E2 -24484.711} C_VEL
LIN {X 0,Y 201.242,Z 457.115,A -85,B 0,C 180,E1 -24486.013,E2 -24486.013} C_VEL
LIN {X 0,Y 204.613,Z 444.857,A -85,B 0,C 180,E1 -24486.962,E2 -24486.962} C_VEL
LIN {X 0,Y 207.27,Z 431.306,A -85,B 0,C 180,E1 -24487.654,E2 -24487.654} C_VEL
LIN {X 0,Y 209.974,Z 410.091,A -85,B 0,C 180,E1 -24488.431,E2 -24488.431} C_VEL
LIN {X 0,Y 208.774,Z 406.961,A -85,B 0,C 180,E1 -24489.779,E2 -24489.779} C_VEL
LIN {X 0,Y 205.785,Z 401.23,A -85,B 0,C 180,E1 -24493.638,E2 -24493.638} C_VEL
LIN {X 0,Y 204.278,Z 398.229,A -85,B 0,C 180,E1 -24496.465,E2 -24496.465} C_VEL
LIN {X 0,Y 202.812,Z 395.979,A -85,B 0,C 180,E1 -24501.648,E2 -24501.648} C_VEL
LIN {X 0,Y 202.907,Z 396.697,A -85,B 0,C 180,E1 -24505.942,E2 -24505.942} C_VEL
LIN {X 0,Y 204.525,Z 401.597,A -85,B 0,C 180,E1 -24511.251,E2 -24511.251} C_VEL
LIN {X 0,Y 206.233,Z 406.332,A -85,B 0,C 180,E1 -24514.212,E2 -24514.212} C_VEL
LIN {X 0,Y 207.949,Z 411.416,A -85,B 0,C 180,E1 -24516.565,E2 -24516.565} C_VEL
LIN {X 0,Y 209.384,Z 416.293,A -85,B 0,C 180,E1 -24518.333,E2 -24518.333} C_VEL
LIN {X 0,Y 206.056,Z 440.893,A -85,B 0,C 180,E1 -24519.249,E2 -24519.249} C_VEL
LIN {X 0,Y 203.107,Z 453.965,A -85,B 0,C 180,E1 -24519.916,E2 -24519.916} C_VEL
LIN {X 0,Y 199.529,Z 465.572,A -85,B 0,C 180,E1 -24520.772,E2 -24520.772} C_VEL
LIN {X 0,Y 194.248,Z 478.865,A -85,B 0,C 180,E1 -24522.122,E2 -24522.122} C_VEL
LIN {X 0,Y 189.161,Z 489.366,A -85,B 0,C 180,E1 -24523.572,E2 -24523.572} C_VEL
LIN {X 0,Y 183.027,Z 499.974,A -85,B 0,C 180,E1 -24525.509,E2 -24525.509} C_VEL
LIN {X 0,Y 177.243,Z 508.68,A -85,B 0,C 180,E1 -24527.616,E2 -24527.616} C_VEL
LIN {X 0,Y 170.749,Z 517.353,A -85,B 0,C 180,E1 -24530.357,E2 -24530.357} C_VEL
LIN {X 0,Y 164.76,Z 524.411,A -85,B 0,C 180,E1 -24533.33,E2 -24533.33} C_VEL
LIN {X 0,Y 159.308,Z 530.13,A -85,B 0,C 180,E1 -24536.532,E2 -24536.532} C_VEL
LIN {X 0,Y 154.502,Z 534.706,A -85,B 0,C 180,E1 -24539.974,E2 -24539.974} C_VEL
LIN {X 0,Y 149.162,Z 539.245,A -85,B 0,C 180,E1 -24544.908,E2 -24544.908} C_VEL
LIN {X 0,Y 144.94,Z 542.2,A -85,B 0,C 180,E1 -24550.157,E2 -24550.157} C_VEL
LIN {X 0,Y 142.612,Z 543.396,A -85,B 0,C 180,E1 -24554.67,E2 -24554.67} C_VEL
LIN {X 0,Y 141.164,Z 543.685,A -85,B 0,C 180,E1 -24556.978,E2 -24556.978} C_VEL
LIN {X 0,Y 137.445,Z 543.334,A -85,B 0,C 180,E1 -24560.756,E2 -24560.756} C_VEL
LIN {X 0,Y 134.728,Z 542.468,A -85,B 0,C 180,E1 -24563.893,E2 -24563.893} C_VEL
LIN {X 0,Y 133.714,Z 541.504,A -85,B 0,C 180,E1 -24566.359,E2 -24566.359} C_VEL
LIN {X 0,Y 133.69,Z 541.13,A -85,B 0,C 180,E1 -24567.194,E2 -24567.194} C_VEL
LIN {X 0,Y 133.982,Z 539.699,A -85,B 0,C 180,E1 -24569.998,E2 -24569.998} C_VEL
LIN {X 0,Y 133.788,Z 536.447,A -85,B 0,C 180,E1 -24574.516,E2 -24574.516} C_VEL
LIN {X 0,Y 134.059,Z 532.055,A -85,B 0,C 180,E1 -24579.047,E2 -24579.047} C_VEL
LIN {X 0,Y 134.875,Z 526.392,A -85,B 0,C 180,E1 -24583.559,E2 -24583.559} C_VEL
LIN {X 0,Y 136.421,Z 519.252,A -85,B 0,C 180,E1 -24588.003,E2 -24588.003} C_VEL
LIN {X 0,Y 138.714,Z 510.301,A -85,B 0,C 180,E1 -24592.331,E2 -24592.331} C_VEL
LIN {X 0,Y 141.143,Z 501.115,A -85,B 0,C 180,E1 -24595.827,E2 -24595.827} C_VEL
LIN {X 0,Y 143.716,Z 490.92,A -85,B 0,C 180,E1 -24598.879,E2 -24598.879} C_VEL
LIN {X 0,Y 146.379,Z 479.751,A -85,B 0,C 180,E1 -24601.473,E2 -24601.473} C_VEL
LIN {X 0,Y 149.009,Z 467.387,A -85,B 0,C 180,E1 -24603.653,E2 -24603.653} C_VEL
LIN {X 0,Y 151.231,Z 454.249,A -85,B 0,C 180,E1 -24605.307,E2 -24605.307} C_VEL
LIN {X 0,Y 152.86,Z 440.429,A -85,B 0,C 180,E1 -24606.498,E2 -24606.498} C_VEL
LIN {X 0,Y 155.936,Z 395.542,A -85,B 0,C 180,E1 -24608.881,E2 -24608.881} C_VEL
LIN {X 0,Y 154.399,Z 379.735,A -85,B 0,C 180,E1 -24610.195,E2 -24610.195} C_VEL
LIN {X 0,Y 147.095,Z 358.555,A -85,B 0,C 180,E1 -24613.104,E2 -24613.104} C_VEL
LIN {X 0,Y 140.941,Z 343.769,A -85,B 0,C 180,E1 -24615.621,E2 -24615.621} C_VEL
LIN {X 0,Y 137.537,Z 337.131,A -85,B 0,C 180,E1 -24616.999,E2 -24616.999} C_VEL
LIN {X 0,Y 136.199,Z 334.484,A -85,B 0,C 180,E1 -24617.568,E2 -24617.568} C_VEL
LIN {X 0,Y 136.028,Z 333.543,A -85,B 0,C 180,E1 -24617.806,E2 -24617.806} C_VEL
LIN {X 0,Y 136.052,Z 333.539,A -85,B 0,C 180,E1 -24621.693,E2 -24621.693} C_VEL
LIN {X 0,Y 136.086,Z 333.531,A -85,B 0,C 180,E1 -24625.717,E2 -24625.717} C_VEL
LIN {X 0,Y 136.142,Z 333.515,A -85,B 0,C 180,E1 -24632.316,E2 -24632.316} C_VEL
LIN {X 0,Y 136.239,Z 333.507,A -85,B 0,C 180,E1 -24638.833,E2 -24638.833} C_VEL
LIN {X 0,Y 136.28,Z 333.508,A -85,B 0,C 180,E1 -24645.058,E2 -24645.058} C_VEL
LIN {X 0,Y 136.493,Z 333.467,A -85,B 0,C 180,E1 -24648.115,E2 -24648.115} C_VEL
LIN {X 0,Y 136.591,Z 333.466,A -85,B 0,C 180,E1 -24651.121,E2 -24651.121} C_VEL
LIN {X 0,Y 137.128,Z 333.384,A -85,B 0,C 180,E1 -24660.001,E2 -24660.001} C_VEL
LIN {X 0,Y 136.545,Z 333.462,A -85,B 0,C 180,E1 -24668.883,E2 -24668.883} C_VEL
LIN {X 0,Y 136.437,Z 333.461,A -85,B 0,C 180,E1 -24671.891,E2 -24671.891} C_VEL
LIN {X 0,Y 136.238,Z 333.511,A -85,B 0,C 180,E1 -24678.031,E2 -24678.031} C_VEL
LIN {X 0,Y 136.192,Z 333.509,A -85,B 0,C 180,E1 -24681.747,E2 -24681.747} C_VEL
LIN {X 0,Y 136.089,Z 333.519,A -85,B 0,C 180,E1 -24688.611,E2 -24688.611} C_VEL
LIN {X 0,Y 136.039,Z 333.537,A -85,B 0,C 180,E1 -24694.631,E2 -24694.631} C_VEL
LIN {X 0,Y 136.025,Z 333.515,A -85,B 0,C 180,E1 -24699.198,E2 -24699.198} C_VEL
LIN {X 0,Y 135.977,Z 333.541,A -85,B 0,C 180,E1 -24703.651,E2 -24703.651} C_VEL
LIN {X 0,Y 135.981,Z 333.545,A -85,B 0,C 180,E1 -24707.79,E2 -24707.79} C_VEL
LIN {X 0,Y 136.019,Z 333.523,A -85,B 0,C 180,E1 -24711.684,E2 -24711.684} C_VEL
LIN {X 0,Y 136.052,Z 333.532,A -85,B 0,C 180,E1 -24715.744,E2 -24715.744} C_VEL
LIN {X 0,Y 136.14,Z 333.526,A -85,B 0,C 180,E1 -24722.317,E2 -24722.317} C_VEL
LIN {X 0,Y 136.234,Z 333.513,A -85,B 0,C 180,E1 -24728.833,E2 -24728.833} C_VEL
LIN {X 0,Y 136.237,Z 333.513,A -85,B 0,C 180,E1 -24735.054,E2 -24735.054} C_VEL
LIN {X 0,Y 136.428,Z 333.489,A -85,B 0,C 180,E1 -24738.179,E2 -24738.179} C_VEL
LIN {X 0,Y 136.539,Z 333.474,A -85,B 0,C 180,E1 -24741.119,E2 -24741.119} C_VEL
LIN {X 0,Y 137.109,Z 333.408,A -85,B 0,C 180,E1 -24750.002,E2 -24750.002} C_VEL
LIN {X 0,Y 137.064,Z 333.68,A -85,B 0,C 180,E1 -24750.369,E2 -24750.369} C_VEL
LIN {X 0,Y 138.232,Z 336.678,A -85,B 0,C 180,E1 -24750.911,E2 -24750.911} C_VEL
LIN {X 0,Y 146.987,Z 354.475,A -85,B 0,C 180,E1 -24754.355,E2 -24754.355} C_VEL
LIN {X 0,Y 155.66,Z 374.981,A -85,B 0,C 180,E1 -24757.507,E2 -24757.507} C_VEL
LIN {X 0,Y 156.832,Z 378.301,A -85,B 0,C 180,E1 -24757.936,E2 -24757.936} C_VEL
LIN {X 0,Y 152.921,Z 431.343,A -85,B 0,C 180,E1 -24760.733,E2 -24760.733} C_VEL
LIN {X 0,Y 151.355,Z 444.747,A -85,B 0,C 180,E1 -24761.945,E2 -24761.945} C_VEL
LIN {X 0,Y 149.428,Z 457.322,A -85,B 0,C 180,E1 -24763.603,E2 -24763.603} C_VEL
LIN {X 0,Y 146.816,Z 470.491,A -85,B 0,C 180,E1 -24765.978,E2 -24765.978} C_VEL
LIN {X 0,Y 144.363,Z 480.999,A -85,B 0,C 180,E1 -24768.449,E2 -24768.449} C_VEL
LIN {X 0,Y 141.785,Z 491.319,A -85,B 0,C 180,E1 -24771.558,E2 -24771.558} C_VEL
LIN {X 0,Y 139.169,Z 501.147,A -85,B 0,C 180,E1 -24775.315,E2 -24775.315} C_VEL
LIN {X 0,Y 136.987,Z 509.357,A -85,B 0,C 180,E1 -24779.286,E2 -24779.286} C_VEL
LIN {X 0,Y 135.294,Z 516.633,A -85,B 0,C 180,E1 -24783.782,E2 -24783.782} C_VEL
LIN {X 0,Y 134.088,Z 522.227,A -85,B 0,C 180,E1 -24788.167,E2 -24788.167} C_VEL
LIN {X 0,Y 133.209,Z 527.25,A -85,B 0,C 180,E1 -24793.306,E2 -24793.306} C_VEL
LIN {X 0,Y 133.049,Z 530.412,A -85,B 0,C 180,E1 -24797.692,E2 -24797.692} C_VEL
LIN {X 0,Y 133.478,Z 532.699,A -85,B 0,C 180,E1 -24802.169,E2 -24802.169} C_VEL
LIN {X 0,Y 134.579,Z 534.126,A -85,B 0,C 180,E1 -24806.676,E2 -24806.676} C_VEL
LIN {X 0,Y 136.985,Z 534.657,A -85,B 0,C 180,E1 -24812.499,E2 -24812.499} C_VEL
LIN {X 0,Y 139.254,Z 534.19,A -85,B 0,C 180,E1 -24816.186,E2 -24816.186} C_VEL
LIN {X 0,Y 142.162,Z 533.009,A -85,B 0,C 180,E1 -24819.938,E2 -24819.938} C_VEL
LIN {X 0,Y 146.202,Z 530.737,A -85,B 0,C 180,E1 -24824.035,E2 -24824.035} C_VEL
LIN {X 0,Y 150.941,Z 527.443,A -85,B 0,C 180,E1 -24827.906,E2 -24827.906} C_VEL
LIN {X 0,Y 157.64,Z 521.842,A -85,B 0,C 180,E1 -24832.313,E2 -24832.313} C_VEL
LIN {X 0,Y 163.962,Z 515.695,A -85,B 0,C 180,E1 -24835.698,E2 -24835.698} C_VEL
LIN {X 0,Y 169.94,Z 509.028,A -85,B 0,C 180,E1 -24838.461,E2 -24838.461} C_VEL
LIN {X 0,Y 176.375,Z 500.831,A -85,B 0,C 180,E1 -24841.023,E2 -24841.023} C_VEL
LIN {X 0,Y 183.045,Z 490.808,A -85,B 0,C 180,E1 -24843.357,E2 -24843.357} C_VEL
LIN {X 0,Y 188.854,Z 480.52,A -85,B 0,C 180,E1 -24845.16,E2 -24845.16} C_VEL
LIN {X 0,Y 193.56,Z 470.623,A -85,B 0,C 180,E1 -24846.515,E2 -24846.515} C_VEL
LIN {X 0,Y 198.203,Z 458.478,A -85,B 0,C 180,E1 -24847.808,E2 -24847.808} C_VEL
LIN {X 0,Y 201.649,Z 446.759,A -85,B 0,C 180,E1 -24848.731,E2 -24848.731} C_VEL
LIN {X 0,Y 204.632,Z 432.833,A -85,B 0,C 180,E1 -24849.447,E2 -24849.447} C_VEL
LIN {X 0,Y 207.143,Z 414.01,A -85,B 0,C 180,E1 -24850.129,E2 -24850.129} C_VEL
LIN {X 0,Y 205.657,Z 411.089,A -85,B 0,C 180,E1 -24851.957,E2 -24851.957} C_VEL
LIN {X 0,Y 204.115,Z 407.732,A -85,B 0,C 180,E1 -24854.343,E2 -24854.343} C_VEL
LIN {X 0,Y 203.064,Z 405.22,A -85,B 0,C 180,E1 -24856.567,E2 -24856.567} C_VEL
LIN {X 0,Y 201.677,Z 403.002,A -85,B 0,C 180,E1 -24861.529,E2 -24861.529} C_VEL
LIN {X 0,Y 201.712,Z 403.631,A -85,B 0,C 180,E1 -24865.66,E2 -24865.66} C_VEL
LIN {X 0,Y 203.032,Z 408.228,A -85,B 0,C 180,E1 -24870.642,E2 -24870.642} C_VEL
LIN {X 0,Y 204.468,Z 412.667,A -85,B 0,C 180,E1 -24873.447,E2 -24873.447} C_VEL
LIN {X 0,Y 205.959,Z 417.614,A -85,B 0,C 180,E1 -24875.783,E2 -24875.783} C_VEL
LIN {X 0,Y 206.567,Z 419.849,A -85,B 0,C 180,E1 -24876.617,E2 -24876.617} C_VEL
LIN {X 0,Y 203.637,Z 440.476,A -85,B 0,C 180,E1 -24877.37,E2 -24877.37} C_VEL
LIN {X 0,Y 200.655,Z 453.236,A -85,B 0,C 180,E1 -24877.994,E2 -24877.994} C_VEL
LIN {X 0,Y 196.499,Z 466.122,A -85,B 0,C 180,E1 -24878.929,E2 -24878.929} C_VEL
LIN {X 0,Y 191.04,Z 479.167,A -85,B 0,C 180,E1 -24880.238,E2 -24880.238} C_VEL
LIN {X 0,Y 185.114,Z 490.643,A -85,B 0,C 180,E1 -24881.833,E2 -24881.833} C_VEL
LIN {X 0,Y 179.387,Z 500.049,A -85,B 0,C 180,E1 -24883.547,E2 -24883.547} C_VEL
LIN {X 0,Y 173.331,Z 508.713,A -85,B 0,C 180,E1 -24885.617,E2 -24885.617} C_VEL
LIN {X 0,Y 166.524,Z 517.272,A -85,B 0,C 180,E1 -24888.338,E2 -24888.338} C_VEL
LIN {X 0,Y 161.19,Z 523.149,A -85,B 0,C 180,E1 -24890.785,E2 -24890.785} C_VEL
LIN {X 0,Y 155.326,Z 529.051,A -85,B 0,C 180,E1 -24893.969,E2 -24893.969} C_VEL
LIN {X 0,Y 149.202,Z 534.484,A -85,B 0,C 180,E1 -24897.98,E2 -24897.98} C_VEL
LIN {X 0,Y 145.434,Z 537.486,A -85,B 0,C 180,E1 -24901.101,E2 -24901.101} C_VEL
LIN {X 0,Y 140.371,Z 541.001,A -85,B 0,C 180,E1 -24906.386,E2 -24906.386} C_VEL
LIN {X 0,Y 136.558,Z 542.929,A -85,B 0,C 180,E1 -24912.012,E2 -24912.012} C_VEL
LIN {X 0,Y 134.455,Z 543.4,A -85,B 0,C 180,E1 -24917.93,E2 -24917.93} C_VEL
LIN {X 0,Y 133.863,Z 543.075,A -85,B 0,C 180,E1 -24920.936,E2 -24920.936} C_VEL
LIN {X 0,Y 133.674,Z 541.221,A -85,B 0,C 180,E1 -24926.985,E2 -24926.985} C_VEL
LIN {X 0,Y 133.69,Z 541.13,A -85,B 0,C 180,E1 -24927.194,E2 -24927.194} C_VEL
LIN {X 0,Y 133.477,Z 540.31,A -85,B 0,C 180,E1 -24928.837,E2 -24928.837} C_VEL
LIN {X 0,Y 132.717,Z 539.322,A -85,B 0,C 180,E1 -24930.444,E2 -24930.444} C_VEL
LIN {X 0,Y 130.334,Z 536.893,A -85,B 0,C 180,E1 -24933.583,E2 -24933.583} C_VEL
LIN {X 0,Y 127.956,Z 533.944,A -85,B 0,C 180,E1 -24936.764,E2 -24936.764} C_VEL
LIN {X 0,Y 127.093,Z 531.398,A -85,B 0,C 180,E1 -24939.193,E2 -24939.193} C_VEL
LIN {X 0,Y 127.111,Z 530.487,A -85,B 0,C 180,E1 -24940.001,E2 -24940.001} C_VEL
LIN {X 0,Y 128.187,Z 523.966,A -85,B 0,C 180,E1 -24945.093,E2 -24945.093} C_VEL
LIN {X 0,Y 130.077,Z 516.326,A -85,B 0,C 180,E1 -24949.734,E2 -24949.734} C_VEL
LIN {X 0,Y 132.127,Z 508.461,A -85,B 0,C 180,E1 -24953.509,E2 -24953.509} C_VEL
LIN {X 0,Y 135.085,Z 497.576,A -85,B 0,C 180,E1 -24957.577,E2 -24957.577} C_VEL
LIN {X 0,Y 137.902,Z 486.968,A -85,B 0,C 180,E1 -24960.637,E2 -24960.637} C_VEL
LIN {X 0,Y 140.756,Z 474.753,A -85,B 0,C 180,E1 -24963.312,E2 -24963.312} C_VEL
LIN {X 0,Y 143.111,Z 463.037,A -85,B 0,C 180,E1 -24965.24,E2 -24965.24} C_VEL
LIN {X 0,Y 145.245,Z 449.912,A -85,B 0,C 180,E1 -24966.781,E2 -24966.781} C_VEL
LIN {X 0,Y 146.748,Z 435.97,A -85,B 0,C 180,E1 -24967.849,E2 -24967.849} C_VEL
LIN {X 0,Y 149.5,Z 395.719,A -85,B 0,C 180,E1 -24970.061,E2 -24970.061} C_VEL
LIN {X 0,Y 148.247,Z 381.996,A -85,B 0,C 180,E1 -24971.234,E2 -24971.234} C_VEL
LIN {X 0,Y 140.979,Z 360.685,A -85,B 0,C 180,E1 -24974.363,E2 -24974.363} C_VEL
LIN {X 0,Y 135.373,Z 347.183,A -85,B 0,C 180,E1 -24976.806,E2 -24976.806} C_VEL
LIN {X 0,Y 131.889,Z 340.549,A -85,B 0,C 180,E1 -24978.299,E2 -24978.299} C_VEL
LIN {X 0,Y 130.065,Z 337.407,A -85,B 0,C 180,E1 -24979.096,E2 -24979.096} C_VEL
LIN {X 0,Y 128.972,Z 334.421,A -85,B 0,C 180,E1 -24979.717,E2 -24979.717} C_VEL
LIN {X 0,Y 128.988,Z 334.418,A -85,B 0,C 180,E1 -24984.81,E2 -24984.81} C_VEL
LIN {X 0,Y 129.029,Z 334.384,A -85,B 0,C 180,E1 -24990.646,E2 -24990.646} C_VEL
LIN {X 0,Y 129.104,Z 334.402,A -85,B 0,C 180,E1 -24997.601,E2 -24997.601} C_VEL
LIN {X 0,Y 129.155,Z 334.39,A -85,B 0,C 180,E1 -25000.945,E2 -25000.945} C_VEL
LIN {X 0,Y 129.412,Z 334.349,A -85,B 0,C 180,E1 -25007.82,E2 -25007.82} C_VEL
LIN {X 0,Y 129.516,Z 334.346,A -85,B 0,C 180,E1 -25010.632,E2 -25010.632} C_VEL
LIN {X 0,Y 130.083,Z 334.26,A -85,B 0,C 180,E1 -25020.001,E2 -25020.001} C_VEL
LIN {X 0,Y 129.468,Z 334.337,A -85,B 0,C 180,E1 -25029.373,E2 -25029.373} C_VEL
LIN {X 0,Y 129.34,Z 334.346,A -85,B 0,C 180,E1 -25032.554,E2 -25032.554} C_VEL
LIN {X 0,Y 129.148,Z 334.392,A -85,B 0,C 180,E1 -25039.058,E2 -25039.058} C_VEL
LIN {X 0,Y 129.104,Z 334.387,A -85,B 0,C 180,E1 -25042.4,E2 -25042.4} C_VEL
LIN {X 0,Y 129.014,Z 334.405,A -85,B 0,C 180,E1 -25049.36,E2 -25049.36} C_VEL
LIN {X 0,Y 128.955,Z 334.417,A -85,B 0,C 180,E1 -25055.169,E2 -25055.169} C_VEL
LIN {X 0,Y 128.922,Z 334.4,A -85,B 0,C 180,E1 -25060.858,E2 -25060.858} C_VEL
LIN {X 0,Y 128.91,Z 334.425,A -85,B 0,C 180,E1 -25065.134,E2 -25065.134} C_VEL
LIN {X 0,Y 128.933,Z 334.417,A -85,B 0,C 180,E1 -25069.742,E2 -25069.742} C_VEL
LIN {X 0,Y 128.955,Z 334.411,A -85,B 0,C 180,E1 -25074.836,E2 -25074.836} C_VEL
LIN {X 0,Y 129.017,Z 334.41,A -85,B 0,C 180,E1 -25080.645,E2 -25080.645} C_VEL
LIN {X 0,Y 129.107,Z 334.403,A -85,B 0,C 180,E1 -25087.604,E2 -25087.604} C_VEL
LIN {X 0,Y 129.161,Z 334.393,A -85,B 0,C 180,E1 -25094.215,E2 -25094.215} C_VEL
LIN {X 0,Y 129.348,Z 334.37,A -85,B 0,C 180,E1 -25097.969,E2 -25097.969} C_VEL
LIN {X 0,Y 129.465,Z 334.355,A -85,B 0,C 180,E1 -25100.629,E2 -25100.629} C_VEL
LIN {X 0,Y 129.804,Z 334.458,A -85,B 0,C 180,E1 -25108.354,E2 -25108.354} C_VEL
LIN {X 0,Y 130.817,Z 337.097,A -85,B 0,C 180,E1 -25108.881,E2 -25108.881} C_VEL
LIN {X 0,Y 132.148,Z 339.02,A -85,B 0,C 180,E1 -25109.43,E2 -25109.43} C_VEL
LIN {X 0,Y 141.507,Z 358.18,A -85,B 0,C 180,E1 -25113.344,E2 -25113.344} C_VEL
LIN {X 0,Y 149.829,Z 378.223,A -85,B 0,C 180,E1 -25116.596,E2 -25116.596} C_VEL
LIN {X 0,Y 150.317,Z 379.502,A -85,B 0,C 180,E1 -25116.779,E2 -25116.779} C_VEL
LIN {X 0,Y 146.465,Z 431.285,A -85,B 0,C 180,E1 -25119.626,E2 -25119.626} C_VEL
LIN {X 0,Y 144.897,Z 444.356,A -85,B 0,C 180,E1 -25120.835,E2 -25120.835} C_VEL
LIN {X 0,Y 142.821,Z 457.354,A -85,B 0,C 180,E1 -25122.585,E2 -25122.585} C_VEL
LIN {X 0,Y 140.39,Z 469.323,A -85,B 0,C 180,E1 -25124.792,E2 -25124.792} C_VEL
LIN {X 0,Y 137.795,Z 480.195,A -85,B 0,C 180,E1 -25127.388,E2 -25127.388} C_VEL
LIN {X 0,Y 135.123,Z 490.61,A -85,B 0,C 180,E1 -25130.572,E2 -25130.572} C_VEL
LIN {X 0,Y 132.251,Z 500.958,A -85,B 0,C 180,E1 -25134.659,E2 -25134.659} C_VEL
LIN {X 0,Y 129.833,Z 509.83,A -85,B 0,C 180,E1 -25139.157,E2 -25139.157} C_VEL
LIN {X 0,Y 128.306,Z 516.151,A -85,B 0,C 180,E1 -25143.215,E2 -25143.215} C_VEL
LIN {X 0,Y 127.127,Z 521.469,A -85,B 0,C 180,E1 -25147.455,E2 -25147.455} C_VEL
LIN {X 0,Y 126.241,Z 525.905,A -85,B 0,C 180,E1 -25151.919,E2 -25151.919} C_VEL
LIN {X 0,Y 125.93,Z 529.434,A -85,B 0,C 180,E1 -25156.514,E2 -25156.514} C_VEL
LIN {X 0,Y 126.392,Z 532.609,A -85,B 0,C 180,E1 -25162.29,E2 -25162.29} C_VEL
LIN {X 0,Y 127.38,Z 534.058,A -85,B 0,C 180,E1 -25166.513,E2 -25166.513} C_VEL
LIN {X 0,Y 128.908,Z 534.841,A -85,B 0,C 180,E1 -25170.731,E2 -25170.731} C_VEL
LIN {X 0,Y 131.386,Z 534.882,A -85,B 0,C 180,E1 -25175.419,E2 -25175.419} C_VEL
LIN {X 0,Y 134.676,Z 534.008,A -85,B 0,C 180,E1 -25179.942,E2 -25179.942} C_VEL
LIN {X 0,Y 140.088,Z 531.429,A -85,B 0,C 180,E1 -25185.472,E2 -25185.472} C_VEL
LIN {X 0,Y 144.159,Z 528.946,A -85,B 0,C 180,E1 -25188.754,E2 -25188.754} C_VEL
LIN {X 0,Y 151.261,Z 523.724,A -85,B 0,C 180,E1 -25193.406,E2 -25193.406} C_VEL
LIN {X 0,Y 157.128,Z 518.686,A -85,B 0,C 180,E1 -25196.502,E2 -25196.502} C_VEL
LIN {X 0,Y 163.224,Z 512.619,A -85,B 0,C 180,E1 -25199.342,E2 -25199.342} C_VEL
LIN {X 0,Y 169.372,Z 505.647,A -85,B 0,C 180,E1 -25201.808,E2 -25201.808} C_VEL
LIN {X 0,Y 176.175,Z 496.818,A -85,B 0,C 180,E1 -25204.194,E2 -25204.194} C_VEL
LIN {X 0,Y 182.206,Z 487.591,A -85,B 0,C 180,E1 -25206.088,E2 -25206.088} C_VEL
LIN {X 0,Y 188.245,Z 476.633,A -85,B 0,C 180,E1 -25207.778,E2 -25207.778} C_VEL
LIN {X 0,Y 193.087,Z 465.91,A -85,B 0,C 180,E1 -25209.055,E2 -25209.055} C_VEL
LIN {X 0,Y 197.277,Z 454.176,A -85,B 0,C 180,E1 -25210.141,E2 -25210.141} C_VEL
LIN {X 0,Y 200.696,Z 441.592,A -85,B 0,C 180,E1 -25210.946,E2 -25210.946} C_VEL
LIN {X 0,Y 203.214,Z 428.015,A -85,B 0,C 180,E1 -25211.532,E2 -25211.532} C_VEL
LIN {X 0,Y 204.458,Z 418.52,A -85,B 0,C 180,E1 -25211.902,E2 -25211.902} C_VEL
LIN {X 0,Y 202.571,Z 414.392,A -85,B 0,C 180,E1 -25214.899,E2 -25214.899} C_VEL
LIN {X 0,Y 201.645,Z 412.044,A -85,B 0,C 180,E1 -25217.105,E2 -25217.105} C_VEL
LIN {X 0,Y 200.509,Z 410.01,A -85,B 0,C 180,E1 -25221.661,E2 -25221.661} C_VEL
LIN {X 0,Y 200.523,Z 410.608,A -85,B 0,C 180,E1 -25225.423,E2 -25225.423} C_VEL
LIN {X 0,Y 201.555,Z 414.786,A -85,B 0,C 180,E1 -25229.967,E2 -25229.967} C_VEL
LIN {X 0,Y 202.783,Z 419.177,A -85,B 0,C 180,E1 -25232.762,E2 -25232.762} C_VEL
LIN {X 0,Y 203.935,Z 423.605,A -85,B 0,C 180,E1 -25234.851,E2 -25234.851} C_VEL
LIN {X 0,Y 201.079,Z 442,A -85,B 0,C 180,E1 -25235.534,E2 -25235.534} C_VEL
LIN {X 0,Y 197.542,Z 455.675,A -85,B 0,C 180,E1 -25236.216,E2 -25236.216} C_VEL
LIN {X 0,Y 192.966,Z 468.695,A -85,B 0,C 180,E1 -25237.182,E2 -25237.182} C_VEL
LIN {X 0,Y 187.368,Z 481.036,A -85,B 0,C 180,E1 -25238.462,E2 -25238.462} C_VEL
LIN {X 0,Y 181.266,Z 492.072,A -85,B 0,C 180,E1 -25240.025,E2 -25240.025} C_VEL
LIN {X 0,Y 174.687,Z 502.071,A -85,B 0,C 180,E1 -25241.9,E2 -25241.9} C_VEL
LIN {X 0,Y 167.238,Z 511.762,A -85,B 0,C 180,E1 -25244.404,E2 -25244.404} C_VEL
LIN {X 0,Y 160.208,Z 519.701,A -85,B 0,C 180,E1 -25247.158,E2 -25247.158} C_VEL
LIN {X 0,Y 153.717,Z 526.159,A -85,B 0,C 180,E1 -25250.2,E2 -25250.2} C_VEL
LIN {X 0,Y 147.722,Z 531.387,A -85,B 0,C 180,E1 -25253.507,E2 -25253.507} C_VEL
LIN {X 0,Y 142.399,Z 535.549,A -85,B 0,C 180,E1 -25257.117,E2 -25257.117} C_VEL
LIN {X 0,Y 139.271,Z 537.805,A -85,B 0,C 180,E1 -25259.692,E2 -25259.692} C_VEL
LIN {X 0,Y 133.883,Z 541.041,A -85,B 0,C 180,E1 -25265.167,E2 -25265.167} C_VEL
LIN {X 0,Y 129.797,Z 542.782,A -85,B 0,C 180,E1 -25271.04,E2 -25271.04} C_VEL
LIN {X 0,Y 128.491,Z 543.114,A -85,B 0,C 180,E1 -25274.127,E2 -25274.127} C_VEL
LIN {X 0,Y 126.85,Z 542.599,A -85,B 0,C 180,E1 -25280.431,E2 -25280.431} C_VEL
LIN {X 0,Y 126.606,Z 540.59,A -85,B 0,C 180,E1 -25286.816,E2 -25286.816} C_VEL
LIN {X 0,Y 126.92,Z 538.993,A -85,B 0,C 180,E1 -25289.998,E2 -25289.998} C_VEL
LIN {X 0,Y 126.732,Z 535.585,A -85,B 0,C 180,E1 -25294.768,E2 -25294.768} C_VEL
LIN {X 0,Y 127.111,Z 530.487,A -85,B 0,C 180,E1 -25300.001,E2 -25300.001} C_VEL
LIN {X 0,Y 126.849,Z 527.691,A -85,B 0,C 180,E1 -25302.332,E2 -25302.332} C_VEL
LIN {X 0,Y 124.969,Z 522.496,A -85,B 0,C 180,E1 -25306.081,E2 -25306.081} C_VEL
LIN {X 0,Y 123.494,Z 516.639,A -85,B 0,C 180,E1 -25309.742,E2 -25309.742} C_VEL
LIN {X 0,Y 123.876,Z 512.796,A -85,B 0,C 180,E1 -25311.84,E2 -25311.84} C_VEL
LIN {X 0,Y 126.106,Z 504.687,A -85,B 0,C 180,E1 -25315.587,E2 -25315.587} C_VEL
LIN {X 0,Y 129.014,Z 494.261,A -85,B 0,C 180,E1 -25319.356,E2 -25319.356} C_VEL
LIN {X 0,Y 131.798,Z 484.034,A -85,B 0,C 180,E1 -25322.222,E2 -25322.222} C_VEL
LIN {X 0,Y 134.498,Z 472.975,A -85,B 0,C 180,E1 -25324.626,E2 -25324.626} C_VEL
LIN {X 0,Y 136.942,Z 460.754,A -85,B 0,C 180,E1 -25326.625,E2 -25326.625} C_VEL
LIN {X 0,Y 139.18,Z 446.754,A -85,B 0,C 180,E1 -25328.209,E2 -25328.209} C_VEL
LIN {X 0,Y 140.437,Z 433.564,A -85,B 0,C 180,E1 -25329.181,E2 -25329.181} C_VEL
LIN {X 0,Y 143.185,Z 396.893,A -85,B 0,C 180,E1 -25331.237,E2 -25331.237} C_VEL
LIN {X 0,Y 142.105,Z 384.189,A -85,B 0,C 180,E1 -25332.375,E2 -25332.375} C_VEL
LIN {X 0,Y 135.267,Z 363.775,A -85,B 0,C 180,E1 -25335.53,E2 -25335.53} C_VEL
LIN {X 0,Y 129.52,Z 349.85,A -85,B 0,C 180,E1 -25338.21,E2 -25338.21} C_VEL
LIN {X 0,Y 125.106,Z 341.823,A -85,B 0,C 180,E1 -25340.25,E2 -25340.25} C_VEL
LIN {X 0,Y 123.389,Z 338.863,A -85,B 0,C 180,E1 -25341.06,E2 -25341.06} C_VEL
LIN {X 0,Y 122.105,Z 336.47,A -85,B 0,C 180,E1 -25341.702,E2 -25341.702} C_VEL
LIN {X 0,Y 121.881,Z 335.303,A -85,B 0,C 180,E1 -25341.944,E2 -25341.944} C_VEL
LIN {X 0,Y 121.941,Z 335.296,A -85,B 0,C 180,E1 -25344.807,E2 -25344.807} C_VEL
LIN {X 0,Y 121.938,Z 335.263,A -85,B 0,C 180,E1 -25349.826,E2 -25349.826} C_VEL
LIN {X 0,Y 121.979,Z 335.294,A -85,B 0,C 180,E1 -25356.215,E2 -25356.215} C_VEL
LIN {X 0,Y 122.044,Z 335.273,A -85,B 0,C 180,E1 -25359.788,E2 -25359.788} C_VEL
LIN {X 0,Y 122.259,Z 335.244,A -85,B 0,C 180,E1 -25366.707,E2 -25366.707} C_VEL
LIN {X 0,Y 122.444,Z 335.223,A -85,B 0,C 180,E1 -25370.085,E2 -25370.085} C_VEL
LIN {X 0,Y 122.602,Z 335.2,A -85,B 0,C 180,E1 -25376.715,E2 -25376.715} C_VEL
LIN {X 0,Y 123.036,Z 335.137,A -85,B 0,C 180,E1 -25380.001,E2 -25380.001} C_VEL
LIN {X 0,Y 122.404,Z 335.228,A -85,B 0,C 180,E1 -25386.797,E2 -25386.797} C_VEL
LIN {X 0,Y 122.319,Z 335.219,A -85,B 0,C 180,E1 -25392.387,E2 -25392.387} C_VEL
LIN {X 0,Y 122.104,Z 335.27,A -85,B 0,C 180,E1 -25396.726,E2 -25396.726} C_VEL
LIN {X 0,Y 122.024,Z 335.267,A -85,B 0,C 180,E1 -25402.856,E2 -25402.856} C_VEL
LIN {X 0,Y 121.936,Z 335.272,A -85,B 0,C 180,E1 -25407.459,E2 -25407.459} C_VEL
LIN {X 0,Y 121.895,Z 335.3,A -85,B 0,C 180,E1 -25411.26,E2 -25411.26} C_VEL
LIN {X 0,Y 121.879,Z 335.294,A -85,B 0,C 180,E1 -25416.172,E2 -25416.172} C_VEL
LIN {X 0,Y 121.862,Z 335.281,A -85,B 0,C 180,E1 -25421.436,E2 -25421.436} C_VEL
LIN {X 0,Y 121.862,Z 335.302,A -85,B 0,C 180,E1 -25428.569,E2 -25428.569} C_VEL
LIN {X 0,Y 121.907,Z 335.288,A -85,B 0,C 180,E1 -25434.797,E2 -25434.797} C_VEL
LIN {X 0,Y 121.926,Z 335.294,A -85,B 0,C 180,E1 -25439.842,E2 -25439.842} C_VEL
LIN {X 0,Y 121.981,Z 335.289,A -85,B 0,C 180,E1 -25446.217,E2 -25446.217} C_VEL
LIN {X 0,Y 122.021,Z 335.282,A -85,B 0,C 180,E1 -25449.785,E2 -25449.785} C_VEL
LIN {X 0,Y 122.192,Z 335.262,A -85,B 0,C 180,E1 -25456.701,E2 -25456.701} C_VEL
LIN {X 0,Y 122.393,Z 335.237,A -85,B 0,C 180,E1 -25460.083,E2 -25460.083} C_VEL
LIN {X 0,Y 122.527,Z 335.319,A -85,B 0,C 180,E1 -25466.096,E2 -25466.096} C_VEL
LIN {X 0,Y 123.537,Z 338.037,A -85,B 0,C 180,E1 -25466.678,E2 -25466.678} C_VEL
LIN {X 0,Y 125.21,Z 340.217,A -85,B 0,C 180,E1 -25467.41,E2 -25467.41} C_VEL
LIN {X 0,Y 128.218,Z 345.655,A -85,B 0,C 180,E1 -25468.823,E2 -25468.823} C_VEL
LIN {X 0,Y 136.329,Z 362.556,A -85,B 0,C 180,E1 -25472.423,E2 -25472.423} C_VEL
LIN {X 0,Y 143.855,Z 380.921,A -85,B 0,C 180,E1 -25475.536,E2 -25475.536} C_VEL
LIN {X 0,Y 140.299,Z 428.733,A -85,B 0,C 180,E1 -25478.243,E2 -25478.243} C_VEL
LIN {X 0,Y 138.678,Z 442.094,A -85,B 0,C 180,E1 -25479.39,E2 -25479.39} C_VEL
LIN {X 0,Y 136.7,Z 455.095,A -85,B 0,C 180,E1 -25481.118,E2 -25481.118} C_VEL
LIN {X 0,Y 134.246,Z 467.014,A -85,B 0,C 180,E1 -25483.242,E2 -25483.242} C_VEL
LIN {X 0,Y 131.544,Z 478.266,A -85,B 0,C 180,E1 -25485.908,E2 -25485.908} C_VEL
LIN {X 0,Y 128.493,Z 489.804,A -85,B 0,C 180,E1 -25489.482,E2 -25489.482} C_VEL
LIN {X 0,Y 125.585,Z 499.959,A -85,B 0,C 180,E1 -25493.579,E2 -25493.579} C_VEL
LIN {X 0,Y 123.078,Z 508.691,A -85,B 0,C 180,E1 -25498.107,E2 -25498.107} C_VEL
LIN {X 0,Y 121.151,Z 516.458,A -85,B 0,C 180,E1 -25503.272,E2 -25503.272} C_VEL
LIN {X 0,Y 119.921,Z 521.856,A -85,B 0,C 180,E1 -25507.85,E2 -25507.85} C_VEL
LIN {X 0,Y 119.066,Z 526.294,A -85,B 0,C 180,E1 -25512.606,E2 -25512.606} C_VEL
LIN {X 0,Y 118.849,Z 529.711,A -85,B 0,C 180,E1 -25517.341,E2 -25517.341} C_VEL
LIN {X 0,Y 118.995,Z 531.34,A -85,B 0,C 180,E1 -25520.159,E2 -25520.159} C_VEL
LIN {X 0,Y 119.856,Z 533.518,A -85,B 0,C 180,E1 -25525.18,E2 -25525.18} C_VEL
LIN {X 0,Y 121.47,Z 534.832,A -85,B 0,C 180,E1 -25530.215,E2 -25530.215} C_VEL
LIN {X 0,Y 124.902,Z 535.238,A -85,B 0,C 180,E1 -25536.803,E2 -25536.803} C_VEL
LIN {X 0,Y 127.834,Z 534.624,A -85,B 0,C 180,E1 -25540.739,E2 -25540.739} C_VEL
LIN {X 0,Y 131.297,Z 533.413,A -85,B 0,C 180,E1 -25544.475,E2 -25544.475} C_VEL
LIN {X 0,Y 137.879,Z 530.094,A -85,B 0,C 180,E1 -25550.032,E2 -25550.032} C_VEL
LIN {X 0,Y 144.657,Z 525.737,A -85,B 0,C 180,E1 -25554.423,E2 -25554.423} C_VEL
LIN {X 0,Y 151.31,Z 520.58,A -85,B 0,C 180,E1 -25557.935,E2 -25557.935} C_VEL
LIN {X 0,Y 158.783,Z 513.772,A -85,B 0,C 180,E1 -25561.269,E2 -25561.269} C_VEL
LIN {X 0,Y 165.057,Z 507.199,A -85,B 0,C 180,E1 -25563.661,E2 -25563.661} C_VEL
LIN {X 0,Y 172.173,Z 498.549,A -85,B 0,C 180,E1 -25566.044,E2 -25566.044} C_VEL
LIN {X 0,Y 178.867,Z 488.978,A -85,B 0,C 180,E1 -25568.021,E2 -25568.021} C_VEL
LIN {X 0,Y 185.405,Z 477.713,A -85,B 0,C 180,E1 -25569.744,E2 -25569.744} C_VEL
LIN {X 0,Y 190.73,Z 466.527,A -85,B 0,C 180,E1 -25571.059,E2 -25571.059} C_VEL
LIN {X 0,Y 195.126,Z 454.884,A -85,B 0,C 180,E1 -25572.105,E2 -25572.105} C_VEL
LIN {X 0,Y 198.659,Z 442.453,A -85,B 0,C 180,E1 -25572.886,E2 -25572.886} C_VEL
LIN {X 0,Y 201.285,Z 428.938,A -85,B 0,C 180,E1 -25573.457,E2 -25573.457} C_VEL
LIN {X 0,Y 202.059,Z 423.585,A -85,B 0,C 180,E1 -25573.615,E2 -25573.615} C_VEL
LIN {X 0,Y 200.957,Z 420.71,A -85,B 0,C 180,E1 -25575.777,E2 -25575.777} C_VEL
LIN {X 0,Y 200.246,Z 418.846,A -85,B 0,C 180,E1 -25577.654,E2 -25577.654} C_VEL
LIN {X 0,Y 199.344,Z 417.003,A -85,B 0,C 180,E1 -25581.794,E2 -25581.794} C_VEL
LIN {X 0,Y 199.327,Z 417.5,A -85,B 0,C 180,E1 -25585.03,E2 -25585.03} C_VEL
LIN {X 0,Y 200.115,Z 421.379,A -85,B 0,C 180,E1 -25589.317,E2 -25589.317} C_VEL
LIN {X 0,Y 201.141,Z 425.679,A -85,B 0,C 180,E1 -25592.081,E2 -25592.081} C_VEL
LIN {X 0,Y 201.604,Z 427.579,A -85,B 0,C 180,E1 -25593.035,E2 -25593.035} C_VEL
LIN {X 0,Y 199.055,Z 442.636,A -85,B 0,C 180,E1 -25593.599,E2 -25593.599} C_VEL
LIN {X 0,Y 195.13,Z 456.792,A -85,B 0,C 180,E1 -25594.294,E2 -25594.294} C_VEL
LIN {X 0,Y 191.098,Z 467.746,A -85,B 0,C 180,E1 -25595.085,E2 -25595.085} C_VEL
LIN {X 0,Y 186.007,Z 478.833,A -85,B 0,C 180,E1 -25596.134,E2 -25596.134} C_VEL
LIN {X 0,Y 179.654,Z 490.197,A -85,B 0,C 180,E1 -25597.609,E2 -25597.609} C_VEL
LIN {X 0,Y 172.808,Z 500.47,A -85,B 0,C 180,E1 -25599.4,E2 -25599.4} C_VEL
LIN {X 0,Y 166.226,Z 508.928,A -85,B 0,C 180,E1 -25601.367,E2 -25601.367} C_VEL
LIN {X 0,Y 158.758,Z 517.276,A -85,B 0,C 180,E1 -25603.996,E2 -25603.996} C_VEL
LIN {X 0,Y 151.637,Z 524.097,A -85,B 0,C 180,E1 -25606.871,E2 -25606.871} C_VEL
LIN {X 0,Y 144.168,Z 530.464,A -85,B 0,C 180,E1 -25610.672,E2 -25610.672} C_VEL
LIN {X 0,Y 138.3,Z 534.753,A -85,B 0,C 180,E1 -25614.24,E2 -25614.24} C_VEL
LIN {X 0,Y 133.201,Z 538.054,A -85,B 0,C 180,E1 -25618.153,E2 -25618.153} C_VEL
LIN {X 0,Y 127.449,Z 541.085,A -85,B 0,C 180,E1 -25623.821,E2 -25623.821} C_VEL
LIN {X 0,Y 123.078,Z 542.612,A -85,B 0,C 180,E1 -25629.962,E2 -25629.962} C_VEL
LIN {X 0,Y 120.567,Z 542.647,A -85,B 0,C 180,E1 -25636.515,E2 -25636.515} C_VEL
LIN {X 0,Y 119.51,Z 541.222,A -85,B 0,C 180,E1 -25643.244,E2 -25643.244} C_VEL
LIN {X 0,Y 119.601,Z 539.559,A -85,B 0,C 180,E1 -25647.37,E2 -25647.37} C_VEL
LIN {X 0,Y 119.775,Z 537.62,A -85,B 0,C 180,E1 -25650.898,E2 -25650.898} C_VEL
LIN {X 0,Y 119.727,Z 533.168,A -85,B 0,C 180,E1 -25656.74,E2 -25656.74} C_VEL
LIN {X 0,Y 120.485,Z 526.964,A -85,B 0,C 180,E1 -25662.633,E2 -25662.633} C_VEL
LIN {X 0,Y 121.912,Z 520.133,A -85,B 0,C 180,E1 -25667.615,E2 -25667.615} C_VEL
LIN {X 0,Y 123.876,Z 512.796,A -85,B 0,C 180,E1 -25671.84,E2 -25671.84} C_VEL
LIN {X 0,Y 124.336,Z 508.796,A -85,B 0,C 180,E1 -25673.834,E2 -25673.834} C_VEL
LIN {X 0,Y 123.446,Z 501.759,A -85,B 0,C 180,E1 -25677.062,E2 -25677.062} C_VEL
LIN {X 0,Y 122.761,Z 494.235,A -85,B 0,C 180,E1 -25680.079,E2 -25680.079} C_VEL
LIN {X 0,Y 123.513,Z 489.432,A -85,B 0,C 180,E1 -25681.655,E2 -25681.655} C_VEL
LIN {X 0,Y 126.6,Z 477.811,A -85,B 0,C 180,E1 -25684.679,E2 -25684.679} C_VEL
LIN {X 0,Y 129.323,Z 466.142,A -85,B 0,C 180,E1 -25686.952,E2 -25686.952} C_VEL
LIN {X 0,Y 131.922,Z 452.29,A -85,B 0,C 180,E1 -25688.873,E2 -25688.873} C_VEL
LIN {X 0,Y 133.567,Z 439.637,A -85,B 0,C 180,E1 -25690.067,E2 -25690.067} C_VEL
LIN {X 0,Y 136.881,Z 397.406,A -85,B 0,C 180,E1 -25692.582,E2 -25692.582} C_VEL
LIN {X 0,Y 135.953,Z 386.252,A -85,B 0,C 180,E1 -25693.638,E2 -25693.638} C_VEL
LIN {X 0,Y 129.683,Z 367.205,A -85,B 0,C 180,E1 -25696.72,E2 -25696.72} C_VEL
LIN {X 0,Y 124.097,Z 353.311,A -85,B 0,C 180,E1 -25699.565,E2 -25699.565} C_VEL
LIN {X 0,Y 118.696,Z 343.589,A -85,B 0,C 180,E1 -25702.233,E2 -25702.233} C_VEL
LIN {X 0,Y 116.449,Z 339.854,A -85,B 0,C 180,E1 -25703.41,E2 -25703.41} C_VEL
LIN {X 0,Y 115.096,Z 337.263,A -85,B 0,C 180,E1 -25704.183,E2 -25704.183} C_VEL
LIN {X 0,Y 114.889,Z 336.175,A -85,B 0,C 180,E1 -25704.47,E2 -25704.47} C_VEL
LIN {X 0,Y 114.865,Z 336.146,A -85,B 0,C 180,E1 -25710.695,E2 -25710.695} C_VEL
LIN {X 0,Y 114.943,Z 336.171,A -85,B 0,C 180,E1 -25716.507,E2 -25716.507} C_VEL
LIN {X 0,Y 115.013,Z 336.158,A -85,B 0,C 180,E1 -25722.211,E2 -25722.211} C_VEL
LIN {X 0,Y 115.28,Z 336.11,A -85,B 0,C 180,E1 -25727.262,E2 -25727.262} C_VEL
LIN {X 0,Y 115.386,Z 336.111,A -85,B 0,C 180,E1 -25733.004,E2 -25733.004} C_VEL
LIN {X 0,Y 115.988,Z 336.014,A -85,B 0,C 180,E1 -25740.001,E2 -25740.001} C_VEL
LIN {X 0,Y 115.358,Z 336.108,A -85,B 0,C 180,E1 -25747,E2 -25747} C_VEL
LIN {X 0,Y 115.251,Z 336.099,A -85,B 0,C 180,E1 -25752.674,E2 -25752.674} C_VEL
LIN {X 0,Y 115.007,Z 336.154,A -85,B 0,C 180,E1 -25757.792,E2 -25757.792} C_VEL
LIN {X 0,Y 114.942,Z 336.141,A -85,B 0,C 180,E1 -25763.493,E2 -25763.493} C_VEL
LIN {X 0,Y 114.852,Z 336.176,A -85,B 0,C 180,E1 -25771.058,E2 -25771.058} C_VEL
LIN {X 0,Y 114.773,Z 336.168,A -85,B 0,C 180,E1 -25777.76,E2 -25777.76} C_VEL
LIN {X 0,Y 114.777,Z 336.173,A -85,B 0,C 180,E1 -25782.715,E2 -25782.715} C_VEL
LIN {X 0,Y 114.784,Z 336.185,A -85,B 0,C 180,E1 -25787.665,E2 -25787.665} C_VEL
LIN {X 0,Y 114.782,Z 336.164,A -85,B 0,C 180,E1 -25792.75,E2 -25792.75} C_VEL
LIN {X 0,Y 114.855,Z 336.179,A -85,B 0,C 180,E1 -25798.946,E2 -25798.946} C_VEL
LIN {X 0,Y 114.946,Z 336.165,A -85,B 0,C 180,E1 -25806.512,E2 -25806.512} C_VEL
LIN {X 0,Y 114.986,Z 336.16,A -85,B 0,C 180,E1 -25812.208,E2 -25812.208} C_VEL
LIN {X 0,Y 115.308,Z 336.122,A -85,B 0,C 180,E1 -25819.466,E2 -25819.466} C_VEL
LIN {X 0,Y 115.396,Z 336.184,A -85,B 0,C 180,E1 -25823.599,E2 -25823.599} C_VEL
LIN {X 0,Y 116.266,Z 338.775,A -85,B 0,C 180,E1 -25824.191,E2 -25824.191} C_VEL
LIN {X 0,Y 118.075,Z 341.34,A -85,B 0,C 180,E1 -25825.11,E2 -25825.11} C_VEL
LIN {X 0,Y 122.731,Z 348.925,A -85,B 0,C 180,E1 -25827.396,E2 -25827.396} C_VEL
LIN {X 0,Y 130.814,Z 366.098,A -85,B 0,C 180,E1 -25831.269,E2 -25831.269} C_VEL
LIN {X 0,Y 137.52,Z 382.725,A -85,B 0,C 180,E1 -25834.239,E2 -25834.239} C_VEL
LIN {X 0,Y 133.704,Z 430.961,A -85,B 0,C 180,E1 -25837.101,E2 -25837.101} C_VEL
LIN {X 0,Y 132.013,Z 443.94,A -85,B 0,C 180,E1 -25838.357,E2 -25838.357} C_VEL
LIN {X 0,Y 129.923,Z 456.416,A -85,B 0,C 180,E1 -25840.128,E2 -25840.128} C_VEL
LIN {X 0,Y 127.227,Z 468.852,A -85,B 0,C 180,E1 -25842.54,E2 -25842.54} C_VEL
LIN {X 0,Y 124.109,Z 481.015,A -85,B 0,C 180,E1 -25845.7,E2 -25845.7} C_VEL
LIN {X 0,Y 121.344,Z 490.856,A -85,B 0,C 180,E1 -25849.015,E2 -25849.015} C_VEL
LIN {X 0,Y 118.497,Z 500.413,A -85,B 0,C 180,E1 -25853.137,E2 -25853.137} C_VEL
LIN {X 0,Y 115.774,Z 509.606,A -85,B 0,C 180,E1 -25858.23,E2 -25858.23} C_VEL
LIN {X 0,Y 113.85,Z 517.25,A -85,B 0,C 180,E1 -25863.753,E2 -25863.753} C_VEL
LIN {X 0,Y 112.63,Z 522.536,A -85,B 0,C 180,E1 -25868.61,E2 -25868.61} C_VEL
LIN {X 0,Y 111.88,Z 526.922,A -85,B 0,C 180,E1 -25873.711,E2 -25873.711} C_VEL
LIN {X 0,Y 111.808,Z 530.383,A -85,B 0,C 180,E1 -25878.966,E2 -25878.966} C_VEL
LIN {X 0,Y 112.884,Z 533.547,A -85,B 0,C 180,E1 -25885.92,E2 -25885.92} C_VEL
LIN {X 0,Y 114.378,Z 534.881,A -85,B 0,C 180,E1 -25890.556,E2 -25890.556} C_VEL
LIN {X 0,Y 116.455,Z 535.494,A -85,B 0,C 180,E1 -25895.01,E2 -25895.01} C_VEL
LIN {X 0,Y 119.687,Z 535.425,A -85,B 0,C 180,E1 -25899.975,E2 -25899.975} C_VEL
LIN {X 0,Y 123.834,Z 534.466,A -85,B 0,C 180,E1 -25904.76,E2 -25904.76} C_VEL
LIN {X 0,Y 130.727,Z 531.679,A -85,B 0,C 180,E1 -25910.718,E2 -25910.718} C_VEL
LIN {X 0,Y 135.632,Z 529.042,A -85,B 0,C 180,E1 -25914.051,E2 -25914.051} C_VEL
LIN {X 0,Y 140.916,Z 525.737,A -85,B 0,C 180,E1 -25917.141,E2 -25917.141} C_VEL
LIN {X 0,Y 148.867,Z 519.858,A -85,B 0,C 180,E1 -25920.965,E2 -25920.965} C_VEL
LIN {X 0,Y 157.072,Z 512.622,A -85,B 0,C 180,E1 -25924.261,E2 -25924.261} C_VEL
LIN {X 0,Y 165.188,Z 504.039,A -85,B 0,C 180,E1 -25927.019,E2 -25927.019} C_VEL
LIN {X 0,Y 173.187,Z 494.084,A -85,B 0,C 180,E1 -25929.341,E2 -25929.341} C_VEL
LIN {X 0,Y 179.816,Z 484.159,A -85,B 0,C 180,E1 -25931.051,E2 -25931.051} C_VEL
LIN {X 0,Y 186.167,Z 472.575,A -85,B 0,C 180,E1 -25932.538,E2 -25932.538} C_VEL
LIN {X 0,Y 191.553,Z 460.203,A -85,B 0,C 180,E1 -25933.753,E2 -25933.753} C_VEL
LIN {X 0,Y 195.441,Z 448.532,A -85,B 0,C 180,E1 -25934.579,E2 -25934.579} C_VEL
LIN {X 0,Y 198.805,Z 434.714,A -85,B 0,C 180,E1 -25935.236,E2 -25935.236} C_VEL
LIN {X 0,Y 199.865,Z 428.361,A -85,B 0,C 180,E1 -25935.485,E2 -25935.485} C_VEL
LIN {X 0,Y 199.025,Z 425.823,A -85,B 0,C 180,E1 -25937.8,E2 -25937.8} C_VEL
LIN {X 0,Y 198.178,Z 424.009,A -85,B 0,C 180,E1 -25941.928,E2 -25941.928} C_VEL
LIN {X 0,Y 198.14,Z 424.507,A -85,B 0,C 180,E1 -25944.779,E2 -25944.779} C_VEL
LIN {X 0,Y 198.731,Z 428.074,A -85,B 0,C 180,E1 -25948.754,E2 -25948.754} C_VEL
LIN {X 0,Y 199.439,Z 431.794,A -85,B 0,C 180,E1 -25951.177,E2 -25951.177} C_VEL
LIN {X 0,Y 196.404,Z 446.647,A -85,B 0,C 180,E1 -25951.755,E2 -25951.755} C_VEL
LIN {X 0,Y 192.347,Z 459.701,A -85,B 0,C 180,E1 -25952.431,E2 -25952.431} C_VEL
LIN {X 0,Y 187.246,Z 472.118,A -85,B 0,C 180,E1 -25953.37,E2 -25953.37} C_VEL
LIN {X 0,Y 181.323,Z 483.615,A -85,B 0,C 180,E1 -25954.548,E2 -25954.548} C_VEL
LIN {X 0,Y 174.838,Z 493.963,A -85,B 0,C 180,E1 -25956.003,E2 -25956.003} C_VEL
LIN {X 0,Y 167.113,Z 504.285,A -85,B 0,C 180,E1 -25957.949,E2 -25957.949} C_VEL
LIN {X 0,Y 159.112,Z 513.458,A -85,B 0,C 180,E1 -25960.363,E2 -25960.363} C_VEL
LIN {X 0,Y 150.23,Z 522.008,A -85,B 0,C 180,E1 -25963.52,E2 -25963.52} C_VEL
LIN {X 0,Y 143.191,Z 527.872,A -85,B 0,C 180,E1 -25966.594,E2 -25966.594} C_VEL
LIN {X 0,Y 136.625,Z 532.61,A -85,B 0,C 180,E1 -25969.982,E2 -25969.982} C_VEL
LIN {X 0,Y 130.507,Z 536.468,A -85,B 0,C 180,E1 -25973.878,E2 -25973.878} C_VEL
LIN {X 0,Y 123.984,Z 539.918,A -85,B 0,C 180,E1 -25979.324,E2 -25979.324} C_VEL
LIN {X 0,Y 118.569,Z 541.927,A -85,B 0,C 180,E1 -25985.484,E2 -25985.484} C_VEL
LIN {X 0,Y 116.414,Z 542.385,A -85,B 0,C 180,E1 -25988.761,E2 -25988.761} C_VEL
LIN {X 0,Y 113.654,Z 542.239,A -85,B 0,C 180,E1 -25995.677,E2 -25995.677} C_VEL
LIN {X 0,Y 112.484,Z 540.595,A -85,B 0,C 180,E1 -26002.819,E2 -26002.819} C_VEL
LIN {X 0,Y 112.558,Z 538.712,A -85,B 0,C 180,E1 -26007.457,E2 -26007.457} C_VEL
LIN {X 0,Y 112.798,Z 537.358,A -85,B 0,C 180,E1 -26009.998,E2 -26009.998} C_VEL
LIN {X 0,Y 112.625,Z 533.587,A -85,B 0,C 180,E1 -26015.369,E2 -26015.369} C_VEL
LIN {X 0,Y 113.077,Z 528.622,A -85,B 0,C 180,E1 -26020.744,E2 -26020.744} C_VEL
LIN {X 0,Y 114.217,Z 522.298,A -85,B 0,C 180,E1 -26026.073,E2 -26026.073} C_VEL
LIN {X 0,Y 116.336,Z 514.352,A -85,B 0,C 180,E1 -26031.249,E2 -26031.249} C_VEL
LIN {X 0,Y 119.171,Z 504.401,A -85,B 0,C 180,E1 -26036.249,E2 -26036.249} C_VEL
LIN {X 0,Y 121.975,Z 494.844,A -85,B 0,C 180,E1 -26039.934,E2 -26039.934} C_VEL
LIN {X 0,Y 123.513,Z 489.432,A -85,B 0,C 180,E1 -26041.655,E2 -26041.655} C_VEL
LIN {X 0,Y 124.29,Z 484.588,A -85,B 0,C 180,E1 -26043.102,E2 -26043.102} C_VEL
LIN {X 0,Y 123.816,Z 476.28,A -85,B 0,C 180,E1 -26045.53,E2 -26045.53} C_VEL
LIN {X 0,Y 123.142,Z 467.537,A -85,B 0,C 180,E1 -26047.762,E2 -26047.762} C_VEL
LIN {X 0,Y 123.606,Z 461.97,A -85,B 0,C 180,E1 -26048.845,E2 -26048.845} C_VEL
LIN {X 0,Y 125.97,Z 448.787,A -85,B 0,C 180,E1 -26050.562,E2 -26050.562} C_VEL
LIN {X 0,Y 127.593,Z 435.196,A -85,B 0,C 180,E1 -26051.722,E2 -26051.722} C_VEL
LIN {X 0,Y 130.575,Z 397.246,A -85,B 0,C 180,E1 -26054.06,E2 -26054.06} C_VEL
LIN {X 0,Y 129.751,Z 387.988,A -85,B 0,C 180,E1 -26055.007,E2 -26055.007} C_VEL
LIN {X 0,Y 123.87,Z 369.867,A -85,B 0,C 180,E1 -26058.172,E2 -26058.172} C_VEL
LIN {X 0,Y 118.765,Z 356.952,A -85,B 0,C 180,E1 -26060.958,E2 -26060.958} C_VEL
LIN {X 0,Y 113.249,Z 347.062,A -85,B 0,C 180,E1 -26063.915,E2 -26063.915} C_VEL
LIN {X 0,Y 109.778,Z 341.128,A -85,B 0,C 180,E1 -26065.966,E2 -26065.966} C_VEL
LIN {X 0,Y 108.202,Z 338.667,A -85,B 0,C 180,E1 -26066.909,E2 -26066.909} C_VEL
LIN {X 0,Y 107.796,Z 337.033,A -85,B 0,C 180,E1 -26067.355,E2 -26067.355} C_VEL
LIN {X 0,Y 107.854,Z 337.054,A -85,B 0,C 180,E1 -26075.815,E2 -26075.815} C_VEL
LIN {X 0,Y 107.904,Z 337.037,A -85,B 0,C 180,E1 -26080.995,E2 -26080.995} C_VEL
LIN {X 0,Y 108.285,Z 336.979,A -85,B 0,C 180,E1 -26088.773,E2 -26088.773} C_VEL
LIN {X 0,Y 108.453,Z 336.964,A -85,B 0,C 180,E1 -26096.285,E2 -26096.285} C_VEL
LIN {X 0,Y 108.913,Z 336.894,A -85,B 0,C 180,E1 -26100.001,E2 -26100.001} C_VEL
LIN {X 0,Y 108.298,Z 336.984,A -85,B 0,C 180,E1 -26107.458,E2 -26107.458} C_VEL
LIN {X 0,Y 108.171,Z 336.981,A -85,B 0,C 180,E1 -26112.961,E2 -26112.961} C_VEL
LIN {X 0,Y 107.9,Z 337.039,A -85,B 0,C 180,E1 -26119.007,E2 -26119.007} C_VEL
LIN {X 0,Y 107.851,Z 337.018,A -85,B 0,C 180,E1 -26124.182,E2 -26124.182} C_VEL
LIN {X 0,Y 107.776,Z 337.059,A -85,B 0,C 180,E1 -26132.04,E2 -26132.04} C_VEL
LIN {X 0,Y 107.681,Z 337.045,A -85,B 0,C 180,E1 -26138.449,E2 -26138.449} C_VEL
LIN {X 0,Y 107.668,Z 337.072,A -85,B 0,C 180,E1 -26145.893,E2 -26145.893} C_VEL
LIN {X 0,Y 107.681,Z 337.05,A -85,B 0,C 180,E1 -26151.557,E2 -26151.557} C_VEL
LIN {X 0,Y 107.791,Z 337.058,A -85,B 0,C 180,E1 -26158.563,E2 -26158.563} C_VEL
LIN {X 0,Y 107.908,Z 337.042,A -85,B 0,C 180,E1 -26167,E2 -26167} C_VEL
LIN {X 0,Y 107.986,Z 337.032,A -85,B 0,C 180,E1 -26174.913,E2 -26174.913} C_VEL
LIN {X 0,Y 108.269,Z 337.11,A -85,B 0,C 180,E1 -26180.728,E2 -26180.728} C_VEL
LIN {X 0,Y 109.199,Z 339.756,A -85,B 0,C 180,E1 -26181.421,E2 -26181.421} C_VEL
LIN {X 0,Y 111.019,Z 342.196,A -85,B 0,C 180,E1 -26182.449,E2 -26182.449} C_VEL
LIN {X 0,Y 117.475,Z 352.649,A -85,B 0,C 180,E1 -26185.982,E2 -26185.982} C_VEL
LIN {X 0,Y 125.306,Z 369.575,A -85,B 0,C 180,E1 -26190.002,E2 -26190.002} C_VEL
LIN {X 0,Y 131.285,Z 384.596,A -85,B 0,C 180,E1 -26192.886,E2 -26192.886} C_VEL
LIN {X 0,Y 127.308,Z 431.466,A -85,B 0,C 180,E1 -26195.754,E2 -26195.754} C_VEL
LIN {X 0,Y 125.547,Z 444.56,A -85,B 0,C 180,E1 -26197.086,E2 -26197.086} C_VEL
LIN {X 0,Y 123.185,Z 457.611,A -85,B 0,C 180,E1 -26199.029,E2 -26199.029} C_VEL
LIN {X 0,Y 120.417,Z 469.762,A -85,B 0,C 180,E1 -26201.547,E2 -26201.547} C_VEL
LIN {X 0,Y 117.403,Z 480.981,A -85,B 0,C 180,E1 -26204.608,E2 -26204.608} C_VEL
LIN {X 0,Y 114.317,Z 491.513,A -85,B 0,C 180,E1 -26208.345,E2 -26208.345} C_VEL
LIN {X 0,Y 111.321,Z 501.088,A -85,B 0,C 180,E1 -26212.751,E2 -26212.751} C_VEL
LIN {X 0,Y 108.641,Z 509.906,A -85,B 0,C 180,E1 -26217.972,E2 -26217.972} C_VEL
LIN {X 0,Y 106.602,Z 517.763,A -85,B 0,C 180,E1 -26224.082,E2 -26224.082} C_VEL
LIN {X 0,Y 105.273,Z 523.376,A -85,B 0,C 180,E1 -26229.734,E2 -26229.734} C_VEL
LIN {X 0,Y 104.685,Z 527.611,A -85,B 0,C 180,E1 -26235.178,E2 -26235.178} C_VEL
LIN {X 0,Y 104.836,Z 530.808,A -85,B 0,C 180,E1 -26240.44,E2 -26240.44} C_VEL
LIN {X 0,Y 105.2,Z 532.195,A -85,B 0,C 180,E1 -26243.293,E2 -26243.293} C_VEL
LIN {X 0,Y 106.598,Z 534.299,A -85,B 0,C 180,E1 -26248.995,E2 -26248.995} C_VEL
LIN {X 0,Y 108.91,Z 535.522,A -85,B 0,C 180,E1 -26254.616,E2 -26254.616} C_VEL
LIN {X 0,Y 112.176,Z 535.869,A -85,B 0,C 180,E1 -26260.018,E2 -26260.018} C_VEL
LIN {X 0,Y 117.388,Z 535.1,A -85,B 0,C 180,E1 -26266.143,E2 -26266.143} C_VEL
LIN {X 0,Y 121.727,Z 533.762,A -85,B 0,C 180,E1 -26270.025,E2 -26270.025} C_VEL
LIN {X 0,Y 129.457,Z 530.418,A -85,B 0,C 180,E1 -26275.525,E2 -26275.525} C_VEL
LIN {X 0,Y 137.566,Z 525.772,A -85,B 0,C 180,E1 -26279.999,E2 -26279.999} C_VEL
LIN {X 0,Y 146.174,Z 519.689,A -85,B 0,C 180,E1 -26283.801,E2 -26283.801} C_VEL
LIN {X 0,Y 154.96,Z 512.252,A -85,B 0,C 180,E1 -26287.012,E2 -26287.012} C_VEL
LIN {X 0,Y 162.47,Z 504.702,A -85,B 0,C 180,E1 -26289.336,E2 -26289.336} C_VEL
LIN {X 0,Y 170.756,Z 494.801,A -85,B 0,C 180,E1 -26291.574,E2 -26291.574} C_VEL
LIN {X 0,Y 177.449,Z 485.232,A -85,B 0,C 180,E1 -26293.163,E2 -26293.163} C_VEL
LIN {X 0,Y 184.464,Z 472.986,A -85,B 0,C 180,E1 -26294.681,E2 -26294.681} C_VEL
LIN {X 0,Y 189.923,Z 461.013,A -85,B 0,C 180,E1 -26295.818,E2 -26295.818} C_VEL
LIN {X 0,Y 194.204,Z 448.692,A -85,B 0,C 180,E1 -26296.645,E2 -26296.645} C_VEL
LIN {X 0,Y 197.618,Z 435.004,A -85,B 0,C 180,E1 -26297.251,E2 -26297.251} C_VEL
LIN {X 0,Y 197.867,Z 433.598,A -85,B 0,C 180,E1 -26297.335,E2 -26297.335} C_VEL
LIN {X 0,Y 197.602,Z 432.619,A -85,B 0,C 180,E1 -26298.3,E2 -26298.3} C_VEL
LIN {X 0,Y 197.003,Z 431.01,A -85,B 0,C 180,E1 -26301.944,E2 -26301.944} C_VEL
LIN {X 0,Y 196.938,Z 431.444,A -85,B 0,C 180,E1 -26304.471,E2 -26304.471} C_VEL
LIN {X 0,Y 197.273,Z 434.76,A -85,B 0,C 180,E1 -26308.167,E2 -26308.167} C_VEL
LIN {X 0,Y 197.486,Z 436.549,A -85,B 0,C 180,E1 -26309.343,E2 -26309.343} C_VEL
LIN {X 0,Y 193.899,Z 450.879,A -85,B 0,C 180,E1 -26309.892,E2 -26309.892} C_VEL
LIN {X 0,Y 189.68,Z 462.902,A -85,B 0,C 180,E1 -26310.542,E2 -26310.542} C_VEL
LIN {X 0,Y 184.331,Z 474.675,A -85,B 0,C 180,E1 -26311.448,E2 -26311.448} C_VEL
LIN {X 0,Y 177.483,Z 486.77,A -85,B 0,C 180,E1 -26312.703,E2 -26312.703} C_VEL
LIN {X 0,Y 170.12,Z 497.519,A -85,B 0,C 180,E1 -26314.284,E2 -26314.284} C_VEL
LIN {X 0,Y 161.547,Z 507.883,A -85,B 0,C 180,E1 -26316.404,E2 -26316.404} C_VEL
LIN {X 0,Y 153.352,Z 516.28,A -85,B 0,C 180,E1 -26318.82,E2 -26318.82} C_VEL
